// TIA Portal V16 export
// export: Created 2021-11-12T13:31:09.8537827Z, ExportSetting WithDefaults, DisplayName Totally Integrated Automation Portal, DisplayVersion V16 Update 3, DisplayName TIA Portal Version Control Interface, DisplayVersion V16 Update 2, DisplayName TIA Portal Openness, DisplayVersion V16 Update 3, DisplayName SINAMICS Startdrive Advanced, DisplayVersion V16 Update 5, DisplayName SINAMICS Startdrive G130, G150, S120, S150, SINAMICS MV, S210, DisplayVersion V16 Update 5, DisplayName SINAMICS Startdrive G110M, G120, G120C, G120D, G120P, G115D, DisplayVersion V16 Update 5, DisplayName STEP 7 Professional, DisplayVersion V16 Update 3, DisplayName STEP 7 Safety, DisplayVersion V16, DisplayName WinCC UA Professional, DisplayVersion V16 Update 3
FUNCTION_BLOCK "Sfty_Outputs"   // FB74, F_LAD
{ S7_Optimized_Access := 'TRUE' }
VERSION : 0.1
// stored: AutoNumber true, IsIECCheckEnabled false, UDAEnableTagReadback false
   VAR
      "SF_100UH01-KF51_A1" : FDBACK;
      "SF_400UH01-KF51_A1" : FDBACK;
      "SF_100UH01-KF52_A1" : FDBACK;
      "SF_100UH01-KF53_A1" : FDBACK;
   END_VAR
   VAR_TEMP
      TB1EstopZ100 : Bool;   // Estop ok zone 100
      TB1EstopZ200 : Bool;   // Estop ok zone 200
      TB1EstopZ300 : Bool;   // Estop ok zone 300
      TB1EstopZ400 : Bool;   // Estop ok zone 400
      TB1FenceZ101 : Bool;   // Doors locked zone 101
      TB1FenceZ102 : Bool;   // Doors locked zone 102
      TB1FenceZ103 : Bool;   // Doors locked zone 103
      TB1FenceZ104 : Bool;   // Doors locked zone 104
      TB1FenceZ105 : Bool;   // Doors locked zone 105
      TB1FenceZ200 : Bool;   // Doors locked zone 200
      TB1FenceZ300 : Bool;   // Doors locked zone 300
      TB1FenceZ400 : Bool;   // Doors locked zone 400
      TB1Bin : Bool;   // Commissioning
   END_VAR
BEGIN

REGION Network 1: *************** Estop ***************
END_REGION

REGION Network 2: All estops in zone 100 ok
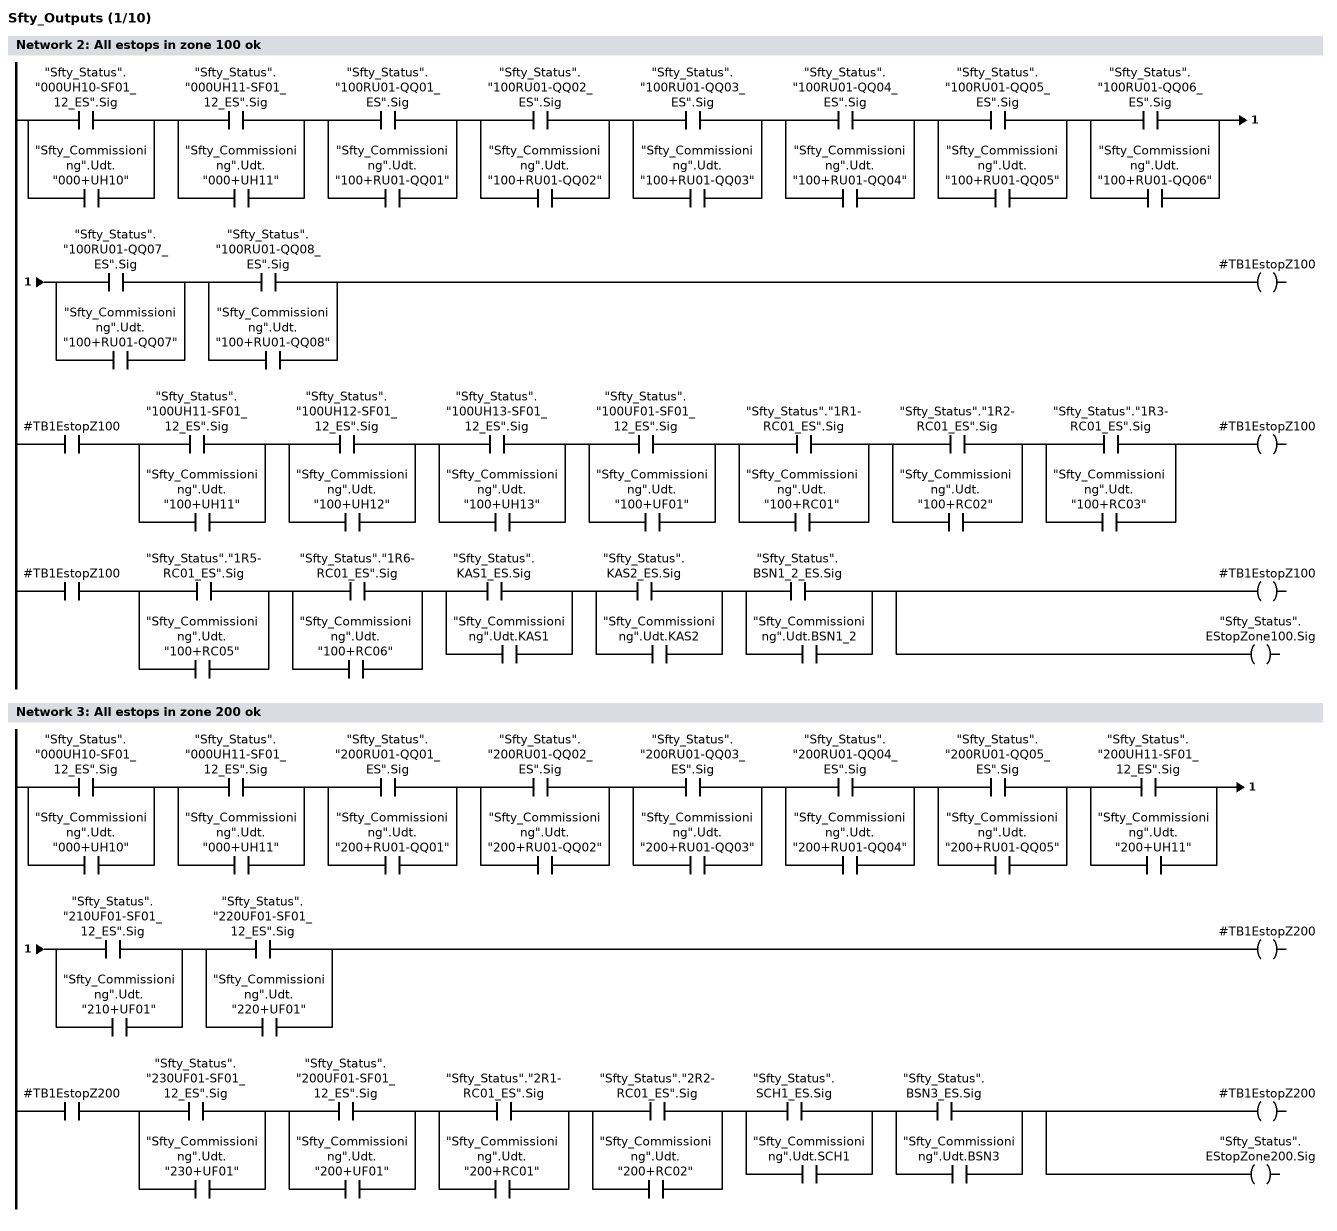
   RUNG wire#powerrail
      Contact( "Sfty_Status"."000UH10-SF01_12_ES".Sig )
      wire#w1
      Contact( "Sfty_Status"."000UH11-SF01_12_ES".Sig )
      wire#w2
      Contact( "Sfty_Status"."100RU01-QQ01_ES".Sig )
      wire#w3
      Contact( "Sfty_Status"."100RU01-QQ02_ES".Sig )
      wire#w4
      Contact( "Sfty_Status"."100RU01-QQ03_ES".Sig )
      wire#w5
      Contact( "Sfty_Status"."100RU01-QQ04_ES".Sig )
      wire#w6
      Contact( "Sfty_Status"."100RU01-QQ05_ES".Sig )
      wire#w7
      Contact( "Sfty_Status"."100RU01-QQ06_ES".Sig )
      wire#w8
      Contact( "Sfty_Status"."100RU01-QQ07_ES".Sig )
      wire#w9
      Contact( "Sfty_Status"."100RU01-QQ08_ES".Sig )
      wire#w10
      Coil( #TB1EstopZ100 )
   END_RUNG
   RUNG wire#powerrail
      Contact( "Sfty_Commissioning".Udt."000+UH10" )
   END_RUNG wire#w1
   RUNG wire#w1
      Contact( "Sfty_Commissioning".Udt."000+UH11" )
   END_RUNG wire#w2
   RUNG wire#w2
      Contact( "Sfty_Commissioning".Udt."100+RU01-QQ01" )
   END_RUNG wire#w3
   RUNG wire#w3
      Contact( "Sfty_Commissioning".Udt."100+RU01-QQ02" )
   END_RUNG wire#w4
   RUNG wire#w4
      Contact( "Sfty_Commissioning".Udt."100+RU01-QQ03" )
   END_RUNG wire#w5
   RUNG wire#w5
      Contact( "Sfty_Commissioning".Udt."100+RU01-QQ04" )
   END_RUNG wire#w6
   RUNG wire#w6
      Contact( "Sfty_Commissioning".Udt."100+RU01-QQ05" )
   END_RUNG wire#w7
   RUNG wire#w7
      Contact( "Sfty_Commissioning".Udt."100+RU01-QQ06" )
   END_RUNG wire#w8
   RUNG wire#w8
      Contact( "Sfty_Commissioning".Udt."100+RU01-QQ07" )
   END_RUNG wire#w9
   RUNG wire#w9
      Contact( "Sfty_Commissioning".Udt."100+RU01-QQ08" )
   END_RUNG wire#w10
   RUNG wire#powerrail
      Contact( #TB1EstopZ100 )
      wire#w11
      Contact( "Sfty_Status"."100UH11-SF01_12_ES".Sig )
      wire#w12
      Contact( "Sfty_Status"."100UH12-SF01_12_ES".Sig )
      wire#w13
      Contact( "Sfty_Status"."100UH13-SF01_12_ES".Sig )
      wire#w14
      Contact( "Sfty_Status"."100UF01-SF01_12_ES".Sig )
      wire#w15
      Contact( "Sfty_Status"."1R1-RC01_ES".Sig )
      wire#w16
      Contact( "Sfty_Status"."1R2-RC01_ES".Sig )
      wire#w17
      Contact( "Sfty_Status"."1R3-RC01_ES".Sig )
      wire#w18
      Coil( #TB1EstopZ100 )
   END_RUNG
   RUNG wire#w11
      Contact( "Sfty_Commissioning".Udt."100+UH11" )
   END_RUNG wire#w12
   RUNG wire#w12
      Contact( "Sfty_Commissioning".Udt."100+UH12" )
   END_RUNG wire#w13
   RUNG wire#w13
      Contact( "Sfty_Commissioning".Udt."100+UH13" )
   END_RUNG wire#w14
   RUNG wire#w14
      Contact( "Sfty_Commissioning".Udt."100+UF01" )
   END_RUNG wire#w15
   RUNG wire#w15
      Contact( "Sfty_Commissioning".Udt."100+RC01" )
   END_RUNG wire#w16
   RUNG wire#w16
      Contact( "Sfty_Commissioning".Udt."100+RC02" )
   END_RUNG wire#w17
   RUNG wire#w17
      Contact( "Sfty_Commissioning".Udt."100+RC03" )
   END_RUNG wire#w18
   RUNG wire#powerrail
      Contact( #TB1EstopZ100 )
      wire#w19
      Contact( "Sfty_Status"."1R5-RC01_ES".Sig )
      wire#w20
      Contact( "Sfty_Status"."1R6-RC01_ES".Sig )
      wire#w21
      Contact( "Sfty_Status".KAS1_ES.Sig )
      wire#w22
      Contact( "Sfty_Status".KAS2_ES.Sig )
      wire#w23
      Contact( "Sfty_Status".BSN1_2_ES.Sig )
      wire#w24
      Coil( #TB1EstopZ100 )
   END_RUNG
   RUNG wire#w19
      Contact( "Sfty_Commissioning".Udt."100+RC05" )
   END_RUNG wire#w20
   RUNG wire#w20
      Contact( "Sfty_Commissioning".Udt."100+RC06" )
   END_RUNG wire#w21
   RUNG wire#w21
      Contact( "Sfty_Commissioning".Udt.KAS1 )
   END_RUNG wire#w22
   RUNG wire#w22
      Contact( "Sfty_Commissioning".Udt.KAS2 )
   END_RUNG wire#w23
   RUNG wire#w23
      Contact( "Sfty_Commissioning".Udt.BSN1_2 )
   END_RUNG wire#w24
   RUNG wire#w24
      Coil( "Sfty_Status".EStopZone100.Sig )
   END_RUNG
   // the same network as SCL:
   #TB1EstopZ100 := ("Sfty_Status"."000UH10-SF01_12_ES".Sig OR "Sfty_Commissioning".Udt."000+UH10") AND ("Sfty_Status"."000UH11-SF01_12_ES".Sig OR "Sfty_Commissioning".Udt."000+UH11") AND ("Sfty_Status"."100RU01-QQ01_ES".Sig OR "Sfty_Commissioning".Udt."100+RU01-QQ01") AND ("Sfty_Status"."100RU01-QQ02_ES".Sig OR "Sfty_Commissioning".Udt."100+RU01-QQ02") AND ("Sfty_Status"."100RU01-QQ03_ES".Sig OR "Sfty_Commissioning".Udt."100+RU01-QQ03") AND ("Sfty_Status"."100RU01-QQ04_ES".Sig OR "Sfty_Commissioning".Udt."100+RU01-QQ04") AND ("Sfty_Status"."100RU01-QQ05_ES".Sig OR "Sfty_Commissioning".Udt."100+RU01-QQ05") AND ("Sfty_Status"."100RU01-QQ06_ES".Sig OR "Sfty_Commissioning".Udt."100+RU01-QQ06") AND ("Sfty_Status"."100RU01-QQ07_ES".Sig OR "Sfty_Commissioning".Udt."100+RU01-QQ07") AND ("Sfty_Status"."100RU01-QQ08_ES".Sig OR "Sfty_Commissioning".Udt."100+RU01-QQ08");
   #TB1EstopZ100 := #TB1EstopZ100 AND ("Sfty_Status"."100UH11-SF01_12_ES".Sig OR "Sfty_Commissioning".Udt."100+UH11") AND ("Sfty_Status"."100UH12-SF01_12_ES".Sig OR "Sfty_Commissioning".Udt."100+UH12") AND ("Sfty_Status"."100UH13-SF01_12_ES".Sig OR "Sfty_Commissioning".Udt."100+UH13") AND ("Sfty_Status"."100UF01-SF01_12_ES".Sig OR "Sfty_Commissioning".Udt."100+UF01") AND ("Sfty_Status"."1R1-RC01_ES".Sig OR "Sfty_Commissioning".Udt."100+RC01") AND ("Sfty_Status"."1R2-RC01_ES".Sig OR "Sfty_Commissioning".Udt."100+RC02") AND ("Sfty_Status"."1R3-RC01_ES".Sig OR "Sfty_Commissioning".Udt."100+RC03");
   #TB1EstopZ100 := #TB1EstopZ100 AND ("Sfty_Status"."1R5-RC01_ES".Sig OR "Sfty_Commissioning".Udt."100+RC05") AND ("Sfty_Status"."1R6-RC01_ES".Sig OR "Sfty_Commissioning".Udt."100+RC06") AND ("Sfty_Status".KAS1_ES.Sig OR "Sfty_Commissioning".Udt.KAS1) AND ("Sfty_Status".KAS2_ES.Sig OR "Sfty_Commissioning".Udt.KAS2) AND ("Sfty_Status".BSN1_2_ES.Sig OR "Sfty_Commissioning".Udt.BSN1_2);
   "Sfty_Status".EStopZone100.Sig := #TB1EstopZ100;
END_REGION

REGION Network 3: All estops in zone 200 ok
   RUNG wire#powerrail
      Contact( "Sfty_Status"."000UH10-SF01_12_ES".Sig )
      wire#w1
      Contact( "Sfty_Status"."000UH11-SF01_12_ES".Sig )
      wire#w2
      Contact( "Sfty_Status"."200RU01-QQ01_ES".Sig )
      wire#w3
      Contact( "Sfty_Status"."200RU01-QQ02_ES".Sig )
      wire#w4
      Contact( "Sfty_Status"."200RU01-QQ03_ES".Sig )
      wire#w5
      Contact( "Sfty_Status"."200RU01-QQ04_ES".Sig )
      wire#w6
      Contact( "Sfty_Status"."200RU01-QQ05_ES".Sig )
      wire#w7
      Contact( "Sfty_Status"."200UH11-SF01_12_ES".Sig )
      wire#w8
      Contact( "Sfty_Status"."210UF01-SF01_12_ES".Sig )
      wire#w9
      Contact( "Sfty_Status"."220UF01-SF01_12_ES".Sig )
      wire#w10
      Coil( #TB1EstopZ200 )
   END_RUNG
   RUNG wire#powerrail
      Contact( "Sfty_Commissioning".Udt."000+UH10" )
   END_RUNG wire#w1
   RUNG wire#w1
      Contact( "Sfty_Commissioning".Udt."000+UH11" )
   END_RUNG wire#w2
   RUNG wire#w2
      Contact( "Sfty_Commissioning".Udt."200+RU01-QQ01" )
   END_RUNG wire#w3
   RUNG wire#w3
      Contact( "Sfty_Commissioning".Udt."200+RU01-QQ02" )
   END_RUNG wire#w4
   RUNG wire#w4
      Contact( "Sfty_Commissioning".Udt."200+RU01-QQ03" )
   END_RUNG wire#w5
   RUNG wire#w5
      Contact( "Sfty_Commissioning".Udt."200+RU01-QQ04" )
   END_RUNG wire#w6
   RUNG wire#w6
      Contact( "Sfty_Commissioning".Udt."200+RU01-QQ05" )
   END_RUNG wire#w7
   RUNG wire#w7
      Contact( "Sfty_Commissioning".Udt."200+UH11" )
   END_RUNG wire#w8
   RUNG wire#w8
      Contact( "Sfty_Commissioning".Udt."210+UF01" )
   END_RUNG wire#w9
   RUNG wire#w9
      Contact( "Sfty_Commissioning".Udt."220+UF01" )
   END_RUNG wire#w10
   RUNG wire#powerrail
      Contact( #TB1EstopZ200 )
      wire#w11
      Contact( "Sfty_Status"."230UF01-SF01_12_ES".Sig )
      wire#w12
      Contact( "Sfty_Status"."200UF01-SF01_12_ES".Sig )
      wire#w13
      Contact( "Sfty_Status"."2R1-RC01_ES".Sig )
      wire#w14
      Contact( "Sfty_Status"."2R2-RC01_ES".Sig )
      wire#w15
      Contact( "Sfty_Status".SCH1_ES.Sig )
      wire#w16
      Contact( "Sfty_Status".BSN3_ES.Sig )
      wire#w17
      Coil( #TB1EstopZ200 )
   END_RUNG
   RUNG wire#w11
      Contact( "Sfty_Commissioning".Udt."230+UF01" )
   END_RUNG wire#w12
   RUNG wire#w12
      Contact( "Sfty_Commissioning".Udt."200+UF01" )
   END_RUNG wire#w13
   RUNG wire#w13
      Contact( "Sfty_Commissioning".Udt."200+RC01" )
   END_RUNG wire#w14
   RUNG wire#w14
      Contact( "Sfty_Commissioning".Udt."200+RC02" )
   END_RUNG wire#w15
   RUNG wire#w15
      Contact( "Sfty_Commissioning".Udt.SCH1 )
   END_RUNG wire#w16
   RUNG wire#w16
      Contact( "Sfty_Commissioning".Udt.BSN3 )
   END_RUNG wire#w17
   RUNG wire#w17
      Coil( "Sfty_Status".EStopZone200.Sig )
   END_RUNG
   // the same network as SCL:
   #TB1EstopZ200 := ("Sfty_Status"."000UH10-SF01_12_ES".Sig OR "Sfty_Commissioning".Udt."000+UH10") AND ("Sfty_Status"."000UH11-SF01_12_ES".Sig OR "Sfty_Commissioning".Udt."000+UH11") AND ("Sfty_Status"."200RU01-QQ01_ES".Sig OR "Sfty_Commissioning".Udt."200+RU01-QQ01") AND ("Sfty_Status"."200RU01-QQ02_ES".Sig OR "Sfty_Commissioning".Udt."200+RU01-QQ02") AND ("Sfty_Status"."200RU01-QQ03_ES".Sig OR "Sfty_Commissioning".Udt."200+RU01-QQ03") AND ("Sfty_Status"."200RU01-QQ04_ES".Sig OR "Sfty_Commissioning".Udt."200+RU01-QQ04") AND ("Sfty_Status"."200RU01-QQ05_ES".Sig OR "Sfty_Commissioning".Udt."200+RU01-QQ05") AND ("Sfty_Status"."200UH11-SF01_12_ES".Sig OR "Sfty_Commissioning".Udt."200+UH11") AND ("Sfty_Status"."210UF01-SF01_12_ES".Sig OR "Sfty_Commissioning".Udt."210+UF01") AND ("Sfty_Status"."220UF01-SF01_12_ES".Sig OR "Sfty_Commissioning".Udt."220+UF01");
   #TB1EstopZ200 := #TB1EstopZ200 AND ("Sfty_Status"."230UF01-SF01_12_ES".Sig OR "Sfty_Commissioning".Udt."230+UF01") AND ("Sfty_Status"."200UF01-SF01_12_ES".Sig OR "Sfty_Commissioning".Udt."200+UF01") AND ("Sfty_Status"."2R1-RC01_ES".Sig OR "Sfty_Commissioning".Udt."200+RC01") AND ("Sfty_Status"."2R2-RC01_ES".Sig OR "Sfty_Commissioning".Udt."200+RC02") AND ("Sfty_Status".SCH1_ES.Sig OR "Sfty_Commissioning".Udt.SCH1) AND ("Sfty_Status".BSN3_ES.Sig OR "Sfty_Commissioning".Udt.BSN3);
   "Sfty_Status".EStopZone200.Sig := #TB1EstopZ200;
END_REGION

REGION Network 4: All estops in zone 300 ok
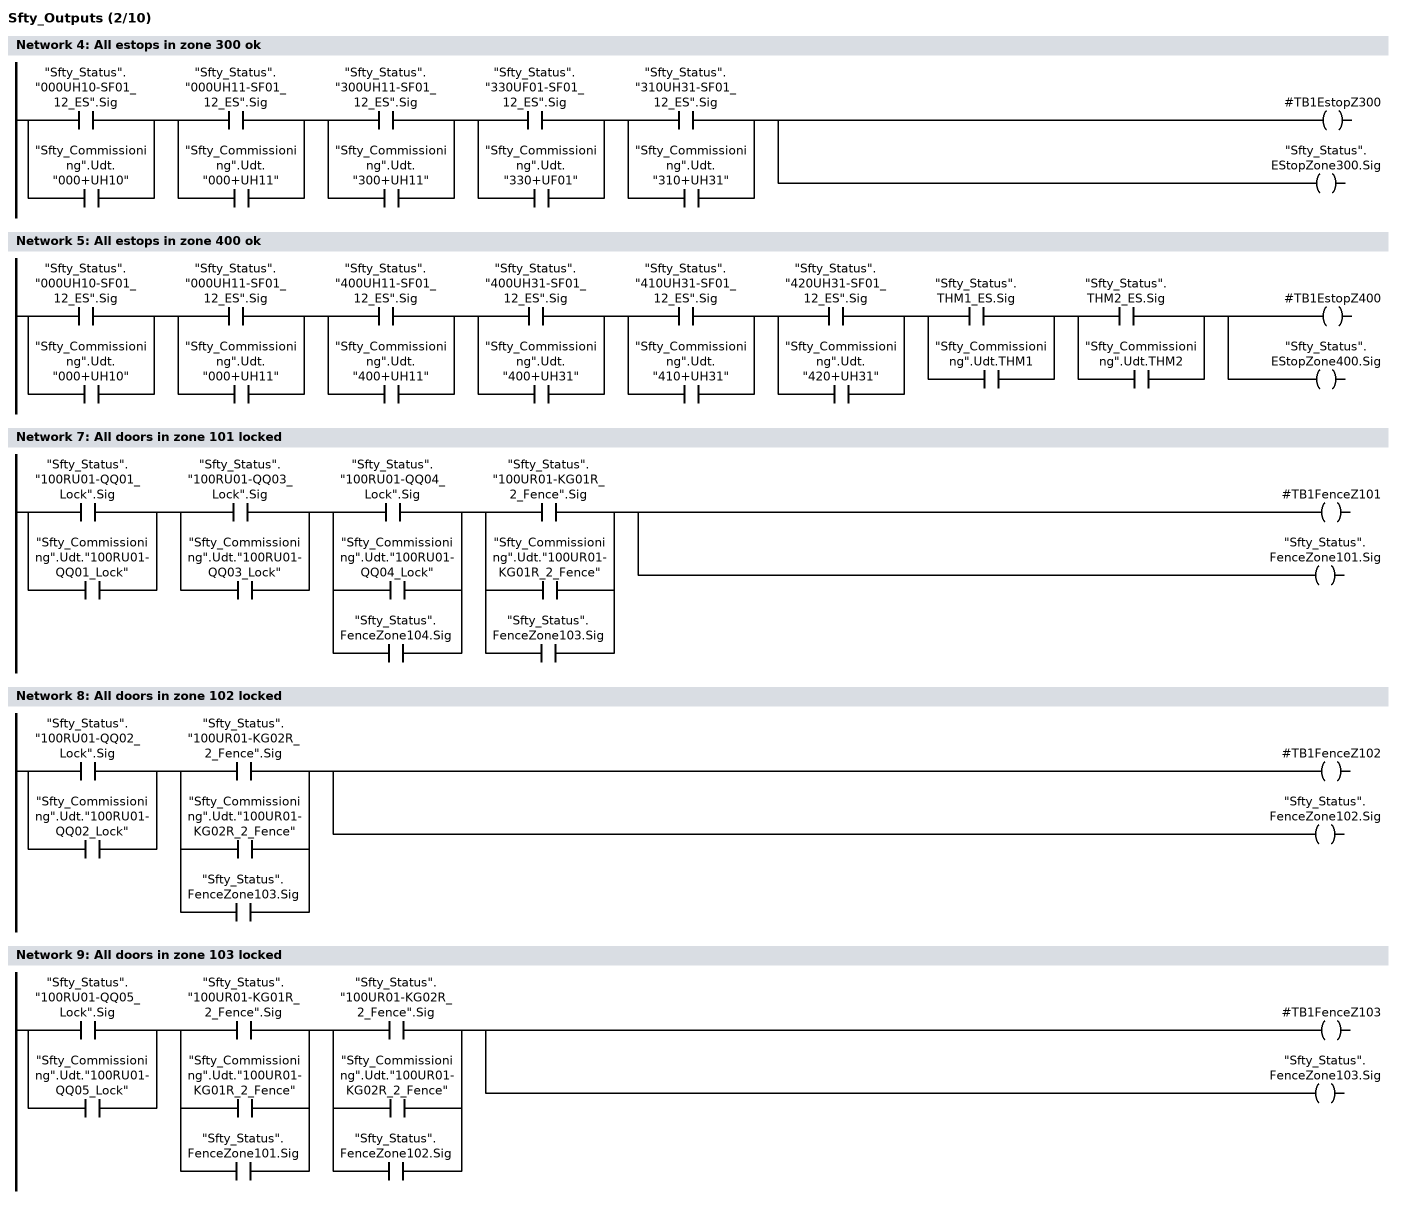
   RUNG wire#powerrail
      Contact( "Sfty_Status"."000UH10-SF01_12_ES".Sig )
      wire#w1
      Contact( "Sfty_Status"."000UH11-SF01_12_ES".Sig )
      wire#w2
      Contact( "Sfty_Status"."300UH11-SF01_12_ES".Sig )
      wire#w3
      Contact( "Sfty_Status"."330UF01-SF01_12_ES".Sig )
      wire#w4
      Contact( "Sfty_Status"."310UH31-SF01_12_ES".Sig )
      wire#w5
      Coil( #TB1EstopZ300 )
   END_RUNG
   RUNG wire#powerrail
      Contact( "Sfty_Commissioning".Udt."000+UH10" )
   END_RUNG wire#w1
   RUNG wire#w1
      Contact( "Sfty_Commissioning".Udt."000+UH11" )
   END_RUNG wire#w2
   RUNG wire#w2
      Contact( "Sfty_Commissioning".Udt."300+UH11" )
   END_RUNG wire#w3
   RUNG wire#w3
      Contact( "Sfty_Commissioning".Udt."330+UF01" )
   END_RUNG wire#w4
   RUNG wire#w4
      Contact( "Sfty_Commissioning".Udt."310+UH31" )
   END_RUNG wire#w5
   RUNG wire#w5
      Coil( "Sfty_Status".EStopZone300.Sig )
   END_RUNG
   // the same network as SCL:
   #TB1EstopZ300 := ("Sfty_Status"."000UH10-SF01_12_ES".Sig OR "Sfty_Commissioning".Udt."000+UH10") AND ("Sfty_Status"."000UH11-SF01_12_ES".Sig OR "Sfty_Commissioning".Udt."000+UH11") AND ("Sfty_Status"."300UH11-SF01_12_ES".Sig OR "Sfty_Commissioning".Udt."300+UH11") AND ("Sfty_Status"."330UF01-SF01_12_ES".Sig OR "Sfty_Commissioning".Udt."330+UF01") AND ("Sfty_Status"."310UH31-SF01_12_ES".Sig OR "Sfty_Commissioning".Udt."310+UH31");
   "Sfty_Status".EStopZone300.Sig := #TB1EstopZ300;
END_REGION

REGION Network 5: All estops in zone 400 ok
   RUNG wire#powerrail
      Contact( "Sfty_Status"."000UH10-SF01_12_ES".Sig )
      wire#w1
      Contact( "Sfty_Status"."000UH11-SF01_12_ES".Sig )
      wire#w2
      Contact( "Sfty_Status"."400UH11-SF01_12_ES".Sig )
      wire#w3
      Contact( "Sfty_Status"."400UH31-SF01_12_ES".Sig )
      wire#w4
      Contact( "Sfty_Status"."410UH31-SF01_12_ES".Sig )
      wire#w5
      Contact( "Sfty_Status"."420UH31-SF01_12_ES".Sig )
      wire#w6
      Contact( "Sfty_Status".THM1_ES.Sig )
      wire#w7
      Contact( "Sfty_Status".THM2_ES.Sig )
      wire#w8
      Coil( #TB1EstopZ400 )
   END_RUNG
   RUNG wire#powerrail
      Contact( "Sfty_Commissioning".Udt."000+UH10" )
   END_RUNG wire#w1
   RUNG wire#w1
      Contact( "Sfty_Commissioning".Udt."000+UH11" )
   END_RUNG wire#w2
   RUNG wire#w2
      Contact( "Sfty_Commissioning".Udt."400+UH11" )
   END_RUNG wire#w3
   RUNG wire#w3
      Contact( "Sfty_Commissioning".Udt."400+UH31" )
   END_RUNG wire#w4
   RUNG wire#w4
      Contact( "Sfty_Commissioning".Udt."410+UH31" )
   END_RUNG wire#w5
   RUNG wire#w5
      Contact( "Sfty_Commissioning".Udt."420+UH31" )
   END_RUNG wire#w6
   RUNG wire#w6
      Contact( "Sfty_Commissioning".Udt.THM1 )
   END_RUNG wire#w7
   RUNG wire#w7
      Contact( "Sfty_Commissioning".Udt.THM2 )
   END_RUNG wire#w8
   RUNG wire#w8
      Coil( "Sfty_Status".EStopZone400.Sig )
   END_RUNG
   // the same network as SCL:
   #TB1EstopZ400 := ("Sfty_Status"."000UH10-SF01_12_ES".Sig OR "Sfty_Commissioning".Udt."000+UH10") AND ("Sfty_Status"."000UH11-SF01_12_ES".Sig OR "Sfty_Commissioning".Udt."000+UH11") AND ("Sfty_Status"."400UH11-SF01_12_ES".Sig OR "Sfty_Commissioning".Udt."400+UH11") AND ("Sfty_Status"."400UH31-SF01_12_ES".Sig OR "Sfty_Commissioning".Udt."400+UH31") AND ("Sfty_Status"."410UH31-SF01_12_ES".Sig OR "Sfty_Commissioning".Udt."410+UH31") AND ("Sfty_Status"."420UH31-SF01_12_ES".Sig OR "Sfty_Commissioning".Udt."420+UH31") AND ("Sfty_Status".THM1_ES.Sig OR "Sfty_Commissioning".Udt.THM1) AND ("Sfty_Status".THM2_ES.Sig OR "Sfty_Commissioning".Udt.THM2);
   "Sfty_Status".EStopZone400.Sig := #TB1EstopZ400;
END_REGION

REGION Network 6: *************** Fence ***************
END_REGION

REGION Network 7: All doors in zone 101 locked
   RUNG wire#powerrail
      Contact( "Sfty_Status"."100RU01-QQ01_Lock".Sig )
      wire#w1
      Contact( "Sfty_Status"."100RU01-QQ03_Lock".Sig )
      wire#w2
      Contact( "Sfty_Status"."100RU01-QQ04_Lock".Sig )
      wire#w3
      Contact( "Sfty_Status"."100UR01-KG01R_2_Fence".Sig )
      wire#w4
      Coil( #TB1FenceZ101 )
   END_RUNG
   RUNG wire#powerrail
      Contact( "Sfty_Commissioning".Udt."100RU01-QQ01_Lock" )
   END_RUNG wire#w1
   RUNG wire#w1
      Contact( "Sfty_Commissioning".Udt."100RU01-QQ03_Lock" )
   END_RUNG wire#w2
   RUNG wire#w2
      Contact( "Sfty_Commissioning".Udt."100RU01-QQ04_Lock" )
   END_RUNG wire#w3
   RUNG wire#w2
      Contact( "Sfty_Status".FenceZone104.Sig )
   END_RUNG wire#w3
   RUNG wire#w3
      Contact( "Sfty_Commissioning".Udt."100UR01-KG01R_2_Fence" )
   END_RUNG wire#w4
   RUNG wire#w3
      Contact( "Sfty_Status".FenceZone103.Sig )
   END_RUNG wire#w4
   RUNG wire#w4
      Coil( "Sfty_Status".FenceZone101.Sig )
   END_RUNG
   // the same network as SCL:
   #TB1FenceZ101 := ("Sfty_Status"."100RU01-QQ01_Lock".Sig OR "Sfty_Commissioning".Udt."100RU01-QQ01_Lock") AND ("Sfty_Status"."100RU01-QQ03_Lock".Sig OR "Sfty_Commissioning".Udt."100RU01-QQ03_Lock") AND ("Sfty_Status"."100RU01-QQ04_Lock".Sig OR "Sfty_Commissioning".Udt."100RU01-QQ04_Lock" OR "Sfty_Status".FenceZone104.Sig) AND ("Sfty_Status"."100UR01-KG01R_2_Fence".Sig OR "Sfty_Commissioning".Udt."100UR01-KG01R_2_Fence" OR "Sfty_Status".FenceZone103.Sig);
   "Sfty_Status".FenceZone101.Sig := #TB1FenceZ101;
END_REGION

REGION Network 8: All doors in zone 102 locked
   RUNG wire#powerrail
      Contact( "Sfty_Status"."100RU01-QQ02_Lock".Sig )
      wire#w1
      Contact( "Sfty_Status"."100UR01-KG02R_2_Fence".Sig )
      wire#w2
      Coil( #TB1FenceZ102 )
   END_RUNG
   RUNG wire#powerrail
      Contact( "Sfty_Commissioning".Udt."100RU01-QQ02_Lock" )
   END_RUNG wire#w1
   RUNG wire#w1
      Contact( "Sfty_Commissioning".Udt."100UR01-KG02R_2_Fence" )
   END_RUNG wire#w2
   RUNG wire#w1
      Contact( "Sfty_Status".FenceZone103.Sig )
   END_RUNG wire#w2
   RUNG wire#w2
      Coil( "Sfty_Status".FenceZone102.Sig )
   END_RUNG
   // the same network as SCL:
   #TB1FenceZ102 := ("Sfty_Status"."100RU01-QQ02_Lock".Sig OR "Sfty_Commissioning".Udt."100RU01-QQ02_Lock") AND ("Sfty_Status"."100UR01-KG02R_2_Fence".Sig OR "Sfty_Commissioning".Udt."100UR01-KG02R_2_Fence" OR "Sfty_Status".FenceZone103.Sig);
   "Sfty_Status".FenceZone102.Sig := #TB1FenceZ102;
END_REGION

REGION Network 9: All doors in zone 103 locked
   RUNG wire#powerrail
      Contact( "Sfty_Status"."100RU01-QQ05_Lock".Sig )
      wire#w1
      Contact( "Sfty_Status"."100UR01-KG01R_2_Fence".Sig )
      wire#w2
      Contact( "Sfty_Status"."100UR01-KG02R_2_Fence".Sig )
      wire#w3
      Coil( #TB1FenceZ103 )
   END_RUNG
   RUNG wire#powerrail
      Contact( "Sfty_Commissioning".Udt."100RU01-QQ05_Lock" )
   END_RUNG wire#w1
   RUNG wire#w1
      Contact( "Sfty_Commissioning".Udt."100UR01-KG01R_2_Fence" )
   END_RUNG wire#w2
   RUNG wire#w1
      Contact( "Sfty_Status".FenceZone101.Sig )
   END_RUNG wire#w2
   RUNG wire#w2
      Contact( "Sfty_Commissioning".Udt."100UR01-KG02R_2_Fence" )
   END_RUNG wire#w3
   RUNG wire#w2
      Contact( "Sfty_Status".FenceZone102.Sig )
   END_RUNG wire#w3
   RUNG wire#w3
      Coil( "Sfty_Status".FenceZone103.Sig )
   END_RUNG
   // the same network as SCL:
   #TB1FenceZ103 := ("Sfty_Status"."100RU01-QQ05_Lock".Sig OR "Sfty_Commissioning".Udt."100RU01-QQ05_Lock") AND ("Sfty_Status"."100UR01-KG01R_2_Fence".Sig OR "Sfty_Commissioning".Udt."100UR01-KG01R_2_Fence" OR "Sfty_Status".FenceZone101.Sig) AND ("Sfty_Status"."100UR01-KG02R_2_Fence".Sig OR "Sfty_Commissioning".Udt."100UR01-KG02R_2_Fence" OR "Sfty_Status".FenceZone102.Sig);
   "Sfty_Status".FenceZone103.Sig := #TB1FenceZ103;
END_REGION

REGION Network 10: All doors in zone 104 locked
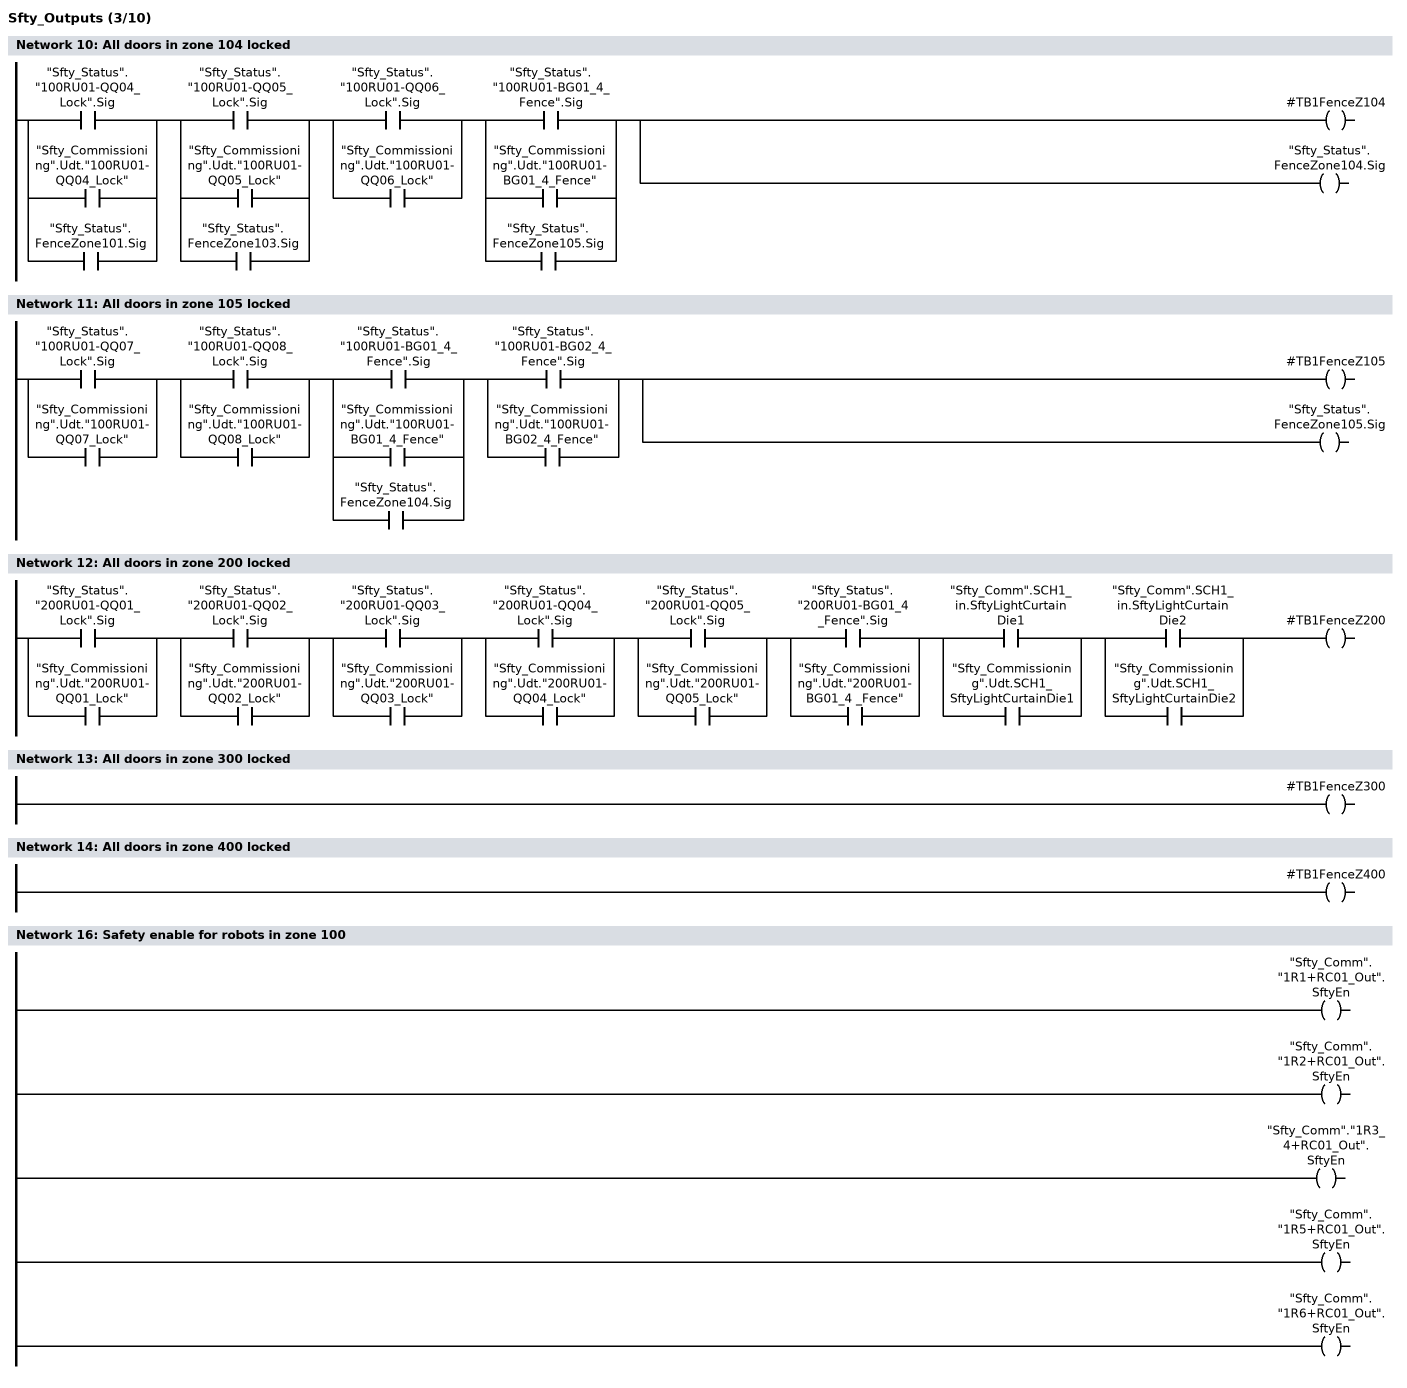
   RUNG wire#powerrail
      Contact( "Sfty_Status"."100RU01-QQ04_Lock".Sig )
      wire#w1
      Contact( "Sfty_Status"."100RU01-QQ05_Lock".Sig )
      wire#w2
      Contact( "Sfty_Status"."100RU01-QQ06_Lock".Sig )
      wire#w3
      Contact( "Sfty_Status"."100RU01-BG01_4_Fence".Sig )
      wire#w4
      Coil( #TB1FenceZ104 )
   END_RUNG
   RUNG wire#powerrail
      Contact( "Sfty_Commissioning".Udt."100RU01-QQ04_Lock" )
   END_RUNG wire#w1
   RUNG wire#powerrail
      Contact( "Sfty_Status".FenceZone101.Sig )
   END_RUNG wire#w1
   RUNG wire#w1
      Contact( "Sfty_Commissioning".Udt."100RU01-QQ05_Lock" )
   END_RUNG wire#w2
   RUNG wire#w1
      Contact( "Sfty_Status".FenceZone103.Sig )
   END_RUNG wire#w2
   RUNG wire#w2
      Contact( "Sfty_Commissioning".Udt."100RU01-QQ06_Lock" )
   END_RUNG wire#w3
   RUNG wire#w3
      Contact( "Sfty_Commissioning".Udt."100RU01-BG01_4_Fence" )
   END_RUNG wire#w4
   RUNG wire#w3
      Contact( "Sfty_Status".FenceZone105.Sig )
   END_RUNG wire#w4
   RUNG wire#w4
      Coil( "Sfty_Status".FenceZone104.Sig )
   END_RUNG
   // the same network as SCL:
   #TB1FenceZ104 := ("Sfty_Status"."100RU01-QQ04_Lock".Sig OR "Sfty_Commissioning".Udt."100RU01-QQ04_Lock" OR "Sfty_Status".FenceZone101.Sig) AND ("Sfty_Status"."100RU01-QQ05_Lock".Sig OR "Sfty_Commissioning".Udt."100RU01-QQ05_Lock" OR "Sfty_Status".FenceZone103.Sig) AND ("Sfty_Status"."100RU01-QQ06_Lock".Sig OR "Sfty_Commissioning".Udt."100RU01-QQ06_Lock") AND ("Sfty_Status"."100RU01-BG01_4_Fence".Sig OR "Sfty_Commissioning".Udt."100RU01-BG01_4_Fence" OR "Sfty_Status".FenceZone105.Sig);
   "Sfty_Status".FenceZone104.Sig := #TB1FenceZ104;
END_REGION

REGION Network 11: All doors in zone 105 locked
   RUNG wire#powerrail
      Contact( "Sfty_Status"."100RU01-QQ07_Lock".Sig )
      wire#w1
      Contact( "Sfty_Status"."100RU01-QQ08_Lock".Sig )
      wire#w2
      Contact( "Sfty_Status"."100RU01-BG01_4_Fence".Sig )
      wire#w3
      Contact( "Sfty_Status"."100RU01-BG02_4_Fence".Sig )
      wire#w4
      Coil( #TB1FenceZ105 )
   END_RUNG
   RUNG wire#powerrail
      Contact( "Sfty_Commissioning".Udt."100RU01-QQ07_Lock" )
   END_RUNG wire#w1
   RUNG wire#w1
      Contact( "Sfty_Commissioning".Udt."100RU01-QQ08_Lock" )
   END_RUNG wire#w2
   RUNG wire#w2
      Contact( "Sfty_Commissioning".Udt."100RU01-BG01_4_Fence" )
   END_RUNG wire#w3
   RUNG wire#w2
      Contact( "Sfty_Status".FenceZone104.Sig )
   END_RUNG wire#w3
   RUNG wire#w3
      Contact( "Sfty_Commissioning".Udt."100RU01-BG02_4_Fence" )
   END_RUNG wire#w4
   RUNG wire#w4
      Coil( "Sfty_Status".FenceZone105.Sig )
   END_RUNG
   // the same network as SCL:
   #TB1FenceZ105 := ("Sfty_Status"."100RU01-QQ07_Lock".Sig OR "Sfty_Commissioning".Udt."100RU01-QQ07_Lock") AND ("Sfty_Status"."100RU01-QQ08_Lock".Sig OR "Sfty_Commissioning".Udt."100RU01-QQ08_Lock") AND ("Sfty_Status"."100RU01-BG01_4_Fence".Sig OR "Sfty_Commissioning".Udt."100RU01-BG01_4_Fence" OR "Sfty_Status".FenceZone104.Sig) AND ("Sfty_Status"."100RU01-BG02_4_Fence".Sig OR "Sfty_Commissioning".Udt."100RU01-BG02_4_Fence");
   "Sfty_Status".FenceZone105.Sig := #TB1FenceZ105;
END_REGION

REGION Network 12: All doors in zone 200 locked
   RUNG wire#powerrail
      Contact( "Sfty_Status"."200RU01-QQ01_Lock".Sig )
      wire#w1
      Contact( "Sfty_Status"."200RU01-QQ02_Lock".Sig )
      wire#w2
      Contact( "Sfty_Status"."200RU01-QQ03_Lock".Sig )
      wire#w3
      Contact( "Sfty_Status"."200RU01-QQ04_Lock".Sig )
      wire#w4
      Contact( "Sfty_Status"."200RU01-QQ05_Lock".Sig )
      wire#w5
      Contact( "Sfty_Status"."200RU01-BG01_4 _Fence".Sig )
      wire#w6
      Contact( "Sfty_Comm".SCH1_in.SftyLightCurtainDie1 )
      wire#w7
      Contact( "Sfty_Comm".SCH1_in.SftyLightCurtainDie2 )
      wire#w8
      Coil( #TB1FenceZ200 )
   END_RUNG
   RUNG wire#powerrail
      Contact( "Sfty_Commissioning".Udt."200RU01-QQ01_Lock" )
   END_RUNG wire#w1
   RUNG wire#w1
      Contact( "Sfty_Commissioning".Udt."200RU01-QQ02_Lock" )
   END_RUNG wire#w2
   RUNG wire#w2
      Contact( "Sfty_Commissioning".Udt."200RU01-QQ03_Lock" )
   END_RUNG wire#w3
   RUNG wire#w3
      Contact( "Sfty_Commissioning".Udt."200RU01-QQ04_Lock" )
   END_RUNG wire#w4
   RUNG wire#w4
      Contact( "Sfty_Commissioning".Udt."200RU01-QQ05_Lock" )
   END_RUNG wire#w5
   RUNG wire#w5
      Contact( "Sfty_Commissioning".Udt."200RU01-BG01_4 _Fence" )
   END_RUNG wire#w6
   RUNG wire#w6
      Contact( "Sfty_Commissioning".Udt.SCH1_SftyLightCurtainDie1 )
   END_RUNG wire#w7
   RUNG wire#w7
      Contact( "Sfty_Commissioning".Udt.SCH1_SftyLightCurtainDie2 )
   END_RUNG wire#w8
   // the same network as SCL:
   #TB1FenceZ200 := ("Sfty_Status"."200RU01-QQ01_Lock".Sig OR "Sfty_Commissioning".Udt."200RU01-QQ01_Lock") AND ("Sfty_Status"."200RU01-QQ02_Lock".Sig OR "Sfty_Commissioning".Udt."200RU01-QQ02_Lock") AND ("Sfty_Status"."200RU01-QQ03_Lock".Sig OR "Sfty_Commissioning".Udt."200RU01-QQ03_Lock") AND ("Sfty_Status"."200RU01-QQ04_Lock".Sig OR "Sfty_Commissioning".Udt."200RU01-QQ04_Lock") AND ("Sfty_Status"."200RU01-QQ05_Lock".Sig OR "Sfty_Commissioning".Udt."200RU01-QQ05_Lock") AND ("Sfty_Status"."200RU01-BG01_4 _Fence".Sig OR "Sfty_Commissioning".Udt."200RU01-BG01_4 _Fence") AND ("Sfty_Comm".SCH1_in.SftyLightCurtainDie1 OR "Sfty_Commissioning".Udt.SCH1_SftyLightCurtainDie1) AND ("Sfty_Comm".SCH1_in.SftyLightCurtainDie2 OR "Sfty_Commissioning".Udt.SCH1_SftyLightCurtainDie2);
END_REGION

REGION Network 13: All doors in zone 300 locked
   RUNG wire#powerrail
      Coil( #TB1FenceZ300 )
   END_RUNG
   // the same network as SCL:
   #TB1FenceZ300 := TRUE;
END_REGION

REGION Network 14: All doors in zone 400 locked
   RUNG wire#powerrail
      Coil( #TB1FenceZ400 )
   END_RUNG
   // the same network as SCL:
   #TB1FenceZ400 := TRUE;
END_REGION

REGION Network 15: *************** Robots section start ***************
END_REGION

REGION Network 16: Safety enable for robots in zone 100
   RUNG wire#powerrail
      Coil( "Sfty_Comm"."1R1+RC01_Out".SftyEn )
   END_RUNG
   RUNG wire#powerrail
      Coil( "Sfty_Comm"."1R2+RC01_Out".SftyEn )
   END_RUNG
   RUNG wire#powerrail
      Coil( "Sfty_Comm"."1R3_4+RC01_Out".SftyEn )
   END_RUNG
   RUNG wire#powerrail
      Coil( "Sfty_Comm"."1R5+RC01_Out".SftyEn )
   END_RUNG
   RUNG wire#powerrail
      Coil( "Sfty_Comm"."1R6+RC01_Out".SftyEn )
   END_RUNG
   // the same network as SCL:
   "Sfty_Comm"."1R1+RC01_Out".SftyEn := TRUE;
   "Sfty_Comm"."1R2+RC01_Out".SftyEn := TRUE;
   "Sfty_Comm"."1R3_4+RC01_Out".SftyEn := TRUE;
   "Sfty_Comm"."1R5+RC01_Out".SftyEn := TRUE;
   "Sfty_Comm"."1R6+RC01_Out".SftyEn := TRUE;
END_REGION

REGION Network 17: Safety enable for robots in zone 200
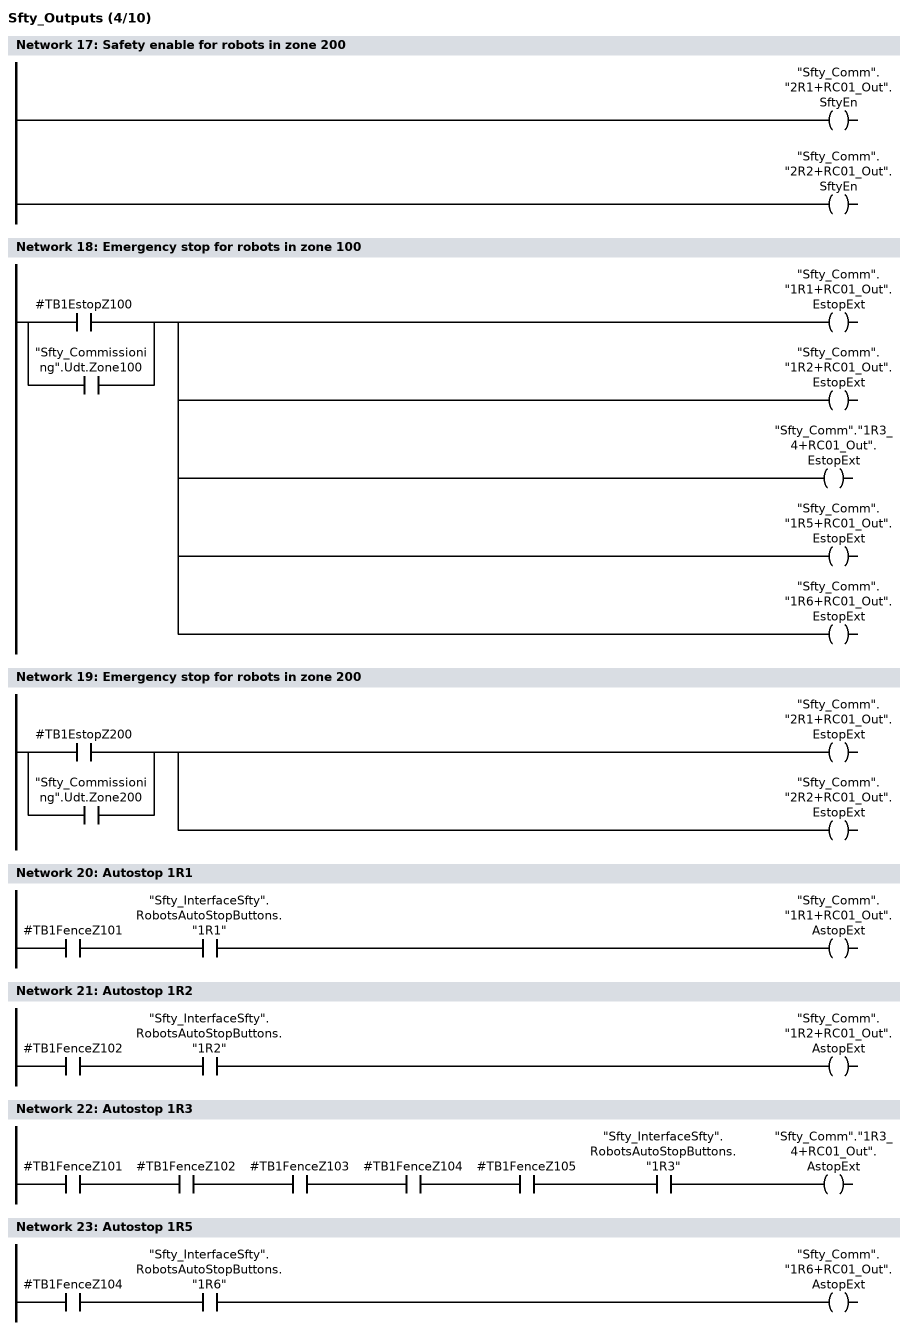
   RUNG wire#powerrail
      Coil( "Sfty_Comm"."2R1+RC01_Out".SftyEn )
   END_RUNG
   RUNG wire#powerrail
      Coil( "Sfty_Comm"."2R2+RC01_Out".SftyEn )
   END_RUNG
   // the same network as SCL:
   "Sfty_Comm"."2R1+RC01_Out".SftyEn := TRUE;
   "Sfty_Comm"."2R2+RC01_Out".SftyEn := TRUE;
END_REGION

REGION Network 18: Emergency stop for robots in zone 100
   RUNG wire#powerrail
      Contact( #TB1EstopZ100 )
      wire#w1
      Coil( "Sfty_Comm"."1R1+RC01_Out".EstopExt )
   END_RUNG
   RUNG wire#powerrail
      Contact( "Sfty_Commissioning".Udt.Zone100 )
   END_RUNG wire#w1
   RUNG wire#w1
      Coil( "Sfty_Comm"."1R2+RC01_Out".EstopExt )
   END_RUNG
   RUNG wire#w1
      Coil( "Sfty_Comm"."1R3_4+RC01_Out".EstopExt )
   END_RUNG
   RUNG wire#w1
      Coil( "Sfty_Comm"."1R5+RC01_Out".EstopExt )
   END_RUNG
   RUNG wire#w1
      Coil( "Sfty_Comm"."1R6+RC01_Out".EstopExt )
   END_RUNG
   // the same network as SCL:
   "Sfty_Comm"."1R1+RC01_Out".EstopExt := #TB1EstopZ100 OR "Sfty_Commissioning".Udt.Zone100;
   "Sfty_Comm"."1R2+RC01_Out".EstopExt := "Sfty_Comm"."1R1+RC01_Out".EstopExt;
   "Sfty_Comm"."1R3_4+RC01_Out".EstopExt := "Sfty_Comm"."1R1+RC01_Out".EstopExt;
   "Sfty_Comm"."1R5+RC01_Out".EstopExt := "Sfty_Comm"."1R1+RC01_Out".EstopExt;
   "Sfty_Comm"."1R6+RC01_Out".EstopExt := "Sfty_Comm"."1R1+RC01_Out".EstopExt;
END_REGION

REGION Network 19: Emergency stop for robots in zone 200
   RUNG wire#powerrail
      Contact( #TB1EstopZ200 )
      wire#w1
      Coil( "Sfty_Comm"."2R1+RC01_Out".EstopExt )
   END_RUNG
   RUNG wire#powerrail
      Contact( "Sfty_Commissioning".Udt.Zone200 )
   END_RUNG wire#w1
   RUNG wire#w1
      Coil( "Sfty_Comm"."2R2+RC01_Out".EstopExt )
   END_RUNG
   // the same network as SCL:
   "Sfty_Comm"."2R1+RC01_Out".EstopExt := #TB1EstopZ200 OR "Sfty_Commissioning".Udt.Zone200;
   "Sfty_Comm"."2R2+RC01_Out".EstopExt := "Sfty_Comm"."2R1+RC01_Out".EstopExt;
END_REGION

REGION Network 20: Autostop 1R1
   RUNG wire#powerrail
      Contact( #TB1FenceZ101 )
      Contact( "Sfty_InterfaceSfty".RobotsAutoStopButtons."1R1" )
      Coil( "Sfty_Comm"."1R1+RC01_Out".AstopExt )
   END_RUNG
   // the same network as SCL:
   "Sfty_Comm"."1R1+RC01_Out".AstopExt := #TB1FenceZ101 AND "Sfty_InterfaceSfty".RobotsAutoStopButtons."1R1";
END_REGION

REGION Network 21: Autostop 1R2
   RUNG wire#powerrail
      Contact( #TB1FenceZ102 )
      Contact( "Sfty_InterfaceSfty".RobotsAutoStopButtons."1R2" )
      Coil( "Sfty_Comm"."1R2+RC01_Out".AstopExt )
   END_RUNG
   // the same network as SCL:
   "Sfty_Comm"."1R2+RC01_Out".AstopExt := #TB1FenceZ102 AND "Sfty_InterfaceSfty".RobotsAutoStopButtons."1R2";
END_REGION

REGION Network 22: Autostop 1R3
   RUNG wire#powerrail
      Contact( #TB1FenceZ101 )
      Contact( #TB1FenceZ102 )
      Contact( #TB1FenceZ103 )
      Contact( #TB1FenceZ104 )
      Contact( #TB1FenceZ105 )
      Contact( "Sfty_InterfaceSfty".RobotsAutoStopButtons."1R3" )
      Coil( "Sfty_Comm"."1R3_4+RC01_Out".AstopExt )
   END_RUNG
   // the same network as SCL:
   "Sfty_Comm"."1R3_4+RC01_Out".AstopExt := #TB1FenceZ101 AND #TB1FenceZ102 AND #TB1FenceZ103 AND #TB1FenceZ104 AND #TB1FenceZ105 AND "Sfty_InterfaceSfty".RobotsAutoStopButtons."1R3";
END_REGION

REGION Network 23: Autostop 1R5
   RUNG wire#powerrail
      Contact( #TB1FenceZ104 )
      Contact( "Sfty_InterfaceSfty".RobotsAutoStopButtons."1R6" )
      Coil( "Sfty_Comm"."1R6+RC01_Out".AstopExt )
   END_RUNG
   // the same network as SCL:
   "Sfty_Comm"."1R6+RC01_Out".AstopExt := #TB1FenceZ104 AND "Sfty_InterfaceSfty".RobotsAutoStopButtons."1R6";
END_REGION

REGION Network 24: Autostop 1R6
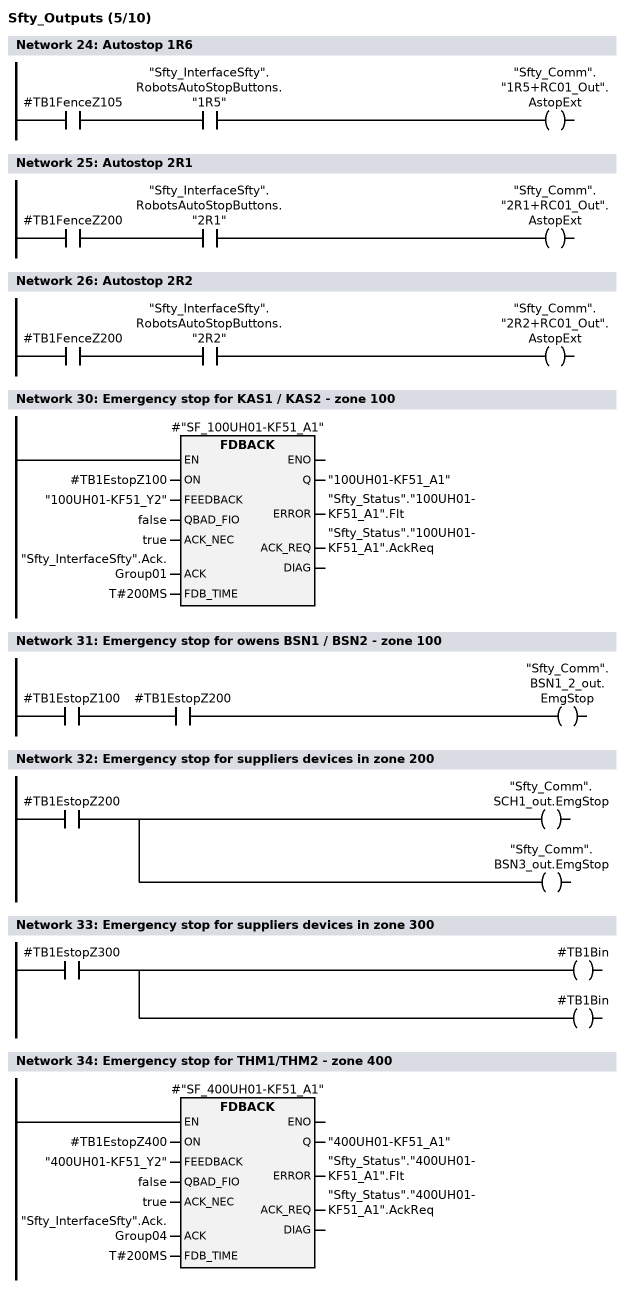
   RUNG wire#powerrail
      Contact( #TB1FenceZ105 )
      Contact( "Sfty_InterfaceSfty".RobotsAutoStopButtons."1R5" )
      Coil( "Sfty_Comm"."1R5+RC01_Out".AstopExt )
   END_RUNG
   // the same network as SCL:
   "Sfty_Comm"."1R5+RC01_Out".AstopExt := #TB1FenceZ105 AND "Sfty_InterfaceSfty".RobotsAutoStopButtons."1R5";
END_REGION

REGION Network 25: Autostop 2R1
   RUNG wire#powerrail
      Contact( #TB1FenceZ200 )
      Contact( "Sfty_InterfaceSfty".RobotsAutoStopButtons."2R1" )
      Coil( "Sfty_Comm"."2R1+RC01_Out".AstopExt )
   END_RUNG
   // the same network as SCL:
   "Sfty_Comm"."2R1+RC01_Out".AstopExt := #TB1FenceZ200 AND "Sfty_InterfaceSfty".RobotsAutoStopButtons."2R1";
END_REGION

REGION Network 26: Autostop 2R2
   RUNG wire#powerrail
      Contact( #TB1FenceZ200 )
      Contact( "Sfty_InterfaceSfty".RobotsAutoStopButtons."2R2" )
      Coil( "Sfty_Comm"."2R2+RC01_Out".AstopExt )
   END_RUNG
   // the same network as SCL:
   "Sfty_Comm"."2R2+RC01_Out".AstopExt := #TB1FenceZ200 AND "Sfty_InterfaceSfty".RobotsAutoStopButtons."2R2";
END_REGION

REGION Network 27: *************** Robots section end ***************
END_REGION

REGION Network 28: *************** Suppliers section start ***************
END_REGION

REGION Network 29: *************** Estop ***************
END_REGION

REGION Network 30: Emergency stop for KAS1 / KAS2 - zone 100
   RUNG wire#powerrail
      #"SF_100UH01-KF51_A1".FDBACK(ON := #TB1EstopZ100, FEEDBACK := "100UH01-KF51_Y2", QBAD_FIO := false, ACK_NEC := true, ACK := "Sfty_InterfaceSfty".Ack.Group01, FDB_TIME := T#200MS, Q => "100UH01-KF51_A1", ERROR => "Sfty_Status"."100UH01-KF51_A1".Flt, ACK_REQ => "Sfty_Status"."100UH01-KF51_A1".AckReq, DIAG =>)
   END_RUNG
   // the same network as SCL:
   #"SF_100UH01-KF51_A1"(ON := #TB1EstopZ100,   // FDBACK
                         FEEDBACK := "100UH01-KF51_Y2",
                         QBAD_FIO := false,
                         ACK_NEC := true,
                         ACK := "Sfty_InterfaceSfty".Ack.Group01,
                         FDB_TIME := T#200MS,
                         Q => "100UH01-KF51_A1",
                         ERROR => "Sfty_Status"."100UH01-KF51_A1".Flt,
                         ACK_REQ => "Sfty_Status"."100UH01-KF51_A1".AckReq);
END_REGION

REGION Network 31: Emergency stop for owens BSN1 / BSN2 - zone 100
   RUNG wire#powerrail
      Contact( #TB1EstopZ100 )
      Contact( #TB1EstopZ200 )
      Coil( "Sfty_Comm".BSN1_2_out.EmgStop )
   END_RUNG
   // the same network as SCL:
   "Sfty_Comm".BSN1_2_out.EmgStop := #TB1EstopZ100 AND #TB1EstopZ200;
END_REGION

REGION Network 32: Emergency stop for suppliers devices in zone 200
   RUNG wire#powerrail
      Contact( #TB1EstopZ200 )
      wire#w1
      Coil( "Sfty_Comm".SCH1_out.EmgStop )
   END_RUNG
   RUNG wire#w1
      Coil( "Sfty_Comm".BSN3_out.EmgStop )
   END_RUNG
   // the same network as SCL:
   "Sfty_Comm".SCH1_out.EmgStop := #TB1EstopZ200;
   "Sfty_Comm".BSN3_out.EmgStop := #TB1EstopZ200;
END_REGION

REGION Network 33: Emergency stop for suppliers devices in zone 300
   RUNG wire#powerrail
      Contact( #TB1EstopZ300 )
      wire#w1
      Coil( #TB1Bin )
   END_RUNG
   RUNG wire#w1
      Coil( #TB1Bin )
   END_RUNG
   // the same network as SCL:
   #TB1Bin := #TB1EstopZ300;
   #TB1Bin := #TB1EstopZ300;
END_REGION

REGION Network 34: Emergency stop for THM1/THM2 - zone 400
   RUNG wire#powerrail
      #"SF_400UH01-KF51_A1".FDBACK(ON := #TB1EstopZ400, FEEDBACK := "400UH01-KF51_Y2", QBAD_FIO := false, ACK_NEC := true, ACK := "Sfty_InterfaceSfty".Ack.Group04, FDB_TIME := T#200MS, Q => "400UH01-KF51_A1", ERROR => "Sfty_Status"."400UH01-KF51_A1".Flt, ACK_REQ => "Sfty_Status"."400UH01-KF51_A1".AckReq, DIAG =>)
   END_RUNG
   // the same network as SCL:
   #"SF_400UH01-KF51_A1"(ON := #TB1EstopZ400,   // FDBACK
                         FEEDBACK := "400UH01-KF51_Y2",
                         QBAD_FIO := false,
                         ACK_NEC := true,
                         ACK := "Sfty_InterfaceSfty".Ack.Group04,
                         FDB_TIME := T#200MS,
                         Q => "400UH01-KF51_A1",
                         ERROR => "Sfty_Status"."400UH01-KF51_A1".Flt,
                         ACK_REQ => "Sfty_Status"."400UH01-KF51_A1".AckReq);
END_REGION

REGION Network 35: Emergency stop for suppliers devices in zone 400
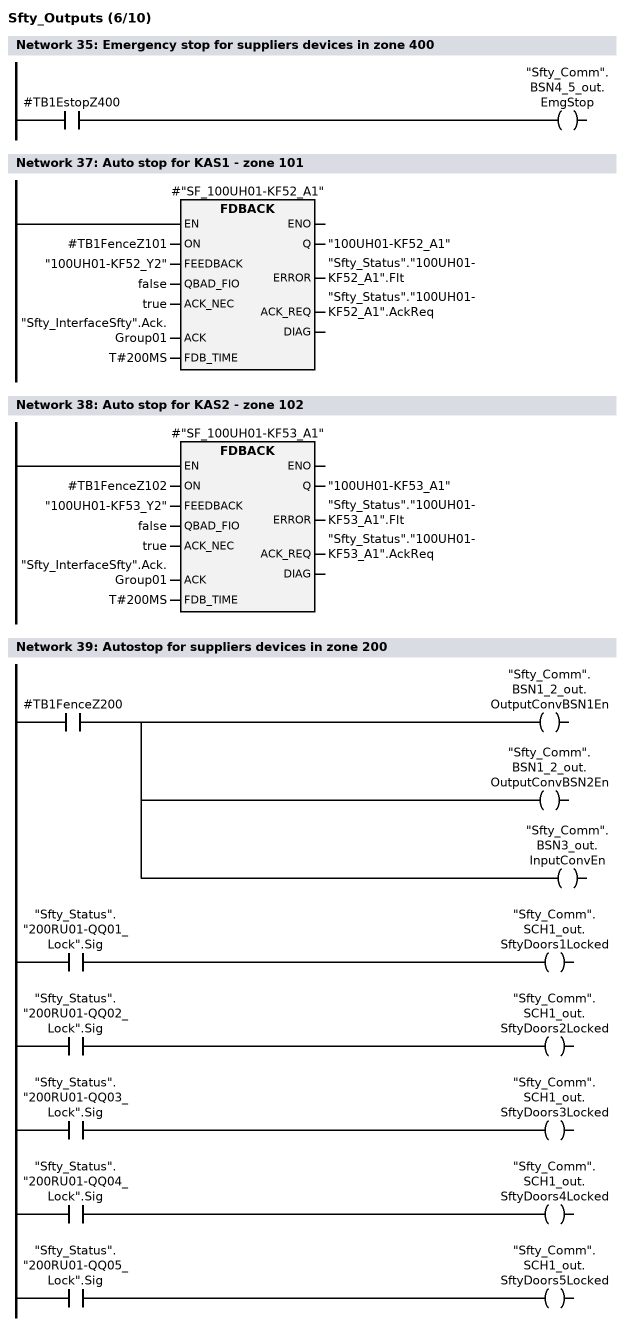
   RUNG wire#powerrail
      Contact( #TB1EstopZ400 )
      Coil( "Sfty_Comm".BSN4_5_out.EmgStop )
   END_RUNG
   // the same network as SCL:
   "Sfty_Comm".BSN4_5_out.EmgStop := #TB1EstopZ400;
END_REGION

REGION Network 36: *************** Auto stop ***************
END_REGION

REGION Network 37: Auto stop for KAS1 - zone 101
   RUNG wire#powerrail
      #"SF_100UH01-KF52_A1".FDBACK(ON := #TB1FenceZ101, FEEDBACK := "100UH01-KF52_Y2", QBAD_FIO := false, ACK_NEC := true, ACK := "Sfty_InterfaceSfty".Ack.Group01, FDB_TIME := T#200MS, Q => "100UH01-KF52_A1", ERROR => "Sfty_Status"."100UH01-KF52_A1".Flt, ACK_REQ => "Sfty_Status"."100UH01-KF52_A1".AckReq, DIAG =>)
   END_RUNG
   // the same network as SCL:
   #"SF_100UH01-KF52_A1"(ON := #TB1FenceZ101,   // FDBACK
                         FEEDBACK := "100UH01-KF52_Y2",
                         QBAD_FIO := false,
                         ACK_NEC := true,
                         ACK := "Sfty_InterfaceSfty".Ack.Group01,
                         FDB_TIME := T#200MS,
                         Q => "100UH01-KF52_A1",
                         ERROR => "Sfty_Status"."100UH01-KF52_A1".Flt,
                         ACK_REQ => "Sfty_Status"."100UH01-KF52_A1".AckReq);
END_REGION

REGION Network 38: Auto stop for KAS2 - zone 102
   RUNG wire#powerrail
      #"SF_100UH01-KF53_A1".FDBACK(ON := #TB1FenceZ102, FEEDBACK := "100UH01-KF53_Y2", QBAD_FIO := false, ACK_NEC := true, ACK := "Sfty_InterfaceSfty".Ack.Group01, FDB_TIME := T#200MS, Q => "100UH01-KF53_A1", ERROR => "Sfty_Status"."100UH01-KF53_A1".Flt, ACK_REQ => "Sfty_Status"."100UH01-KF53_A1".AckReq, DIAG =>)
   END_RUNG
   // the same network as SCL:
   #"SF_100UH01-KF53_A1"(ON := #TB1FenceZ102,   // FDBACK
                         FEEDBACK := "100UH01-KF53_Y2",
                         QBAD_FIO := false,
                         ACK_NEC := true,
                         ACK := "Sfty_InterfaceSfty".Ack.Group01,
                         FDB_TIME := T#200MS,
                         Q => "100UH01-KF53_A1",
                         ERROR => "Sfty_Status"."100UH01-KF53_A1".Flt,
                         ACK_REQ => "Sfty_Status"."100UH01-KF53_A1".AckReq);
END_REGION

REGION Network 39: Autostop for suppliers devices in zone 200
   RUNG wire#powerrail
      Contact( #TB1FenceZ200 )
      wire#w1
      Coil( "Sfty_Comm".BSN1_2_out.OutputConvBSN1En )
   END_RUNG
   RUNG wire#w1
      Coil( "Sfty_Comm".BSN1_2_out.OutputConvBSN2En )
   END_RUNG
   RUNG wire#w1
      Coil( "Sfty_Comm".BSN3_out.InputConvEn )
   END_RUNG
   RUNG wire#powerrail
      Contact( "Sfty_Status"."200RU01-QQ01_Lock".Sig )
      Coil( "Sfty_Comm".SCH1_out.SftyDoors1Locked )
   END_RUNG
   RUNG wire#powerrail
      Contact( "Sfty_Status"."200RU01-QQ02_Lock".Sig )
      Coil( "Sfty_Comm".SCH1_out.SftyDoors2Locked )
   END_RUNG
   RUNG wire#powerrail
      Contact( "Sfty_Status"."200RU01-QQ03_Lock".Sig )
      Coil( "Sfty_Comm".SCH1_out.SftyDoors3Locked )
   END_RUNG
   RUNG wire#powerrail
      Contact( "Sfty_Status"."200RU01-QQ04_Lock".Sig )
      Coil( "Sfty_Comm".SCH1_out.SftyDoors4Locked )
   END_RUNG
   RUNG wire#powerrail
      Contact( "Sfty_Status"."200RU01-QQ05_Lock".Sig )
      Coil( "Sfty_Comm".SCH1_out.SftyDoors5Locked )
   END_RUNG
   // the same network as SCL:
   "Sfty_Comm".BSN1_2_out.OutputConvBSN1En := #TB1FenceZ200;
   "Sfty_Comm".BSN1_2_out.OutputConvBSN2En := #TB1FenceZ200;
   "Sfty_Comm".BSN3_out.InputConvEn := #TB1FenceZ200;
   "Sfty_Comm".SCH1_out.SftyDoors1Locked := "Sfty_Status"."200RU01-QQ01_Lock".Sig;
   "Sfty_Comm".SCH1_out.SftyDoors2Locked := "Sfty_Status"."200RU01-QQ02_Lock".Sig;
   "Sfty_Comm".SCH1_out.SftyDoors3Locked := "Sfty_Status"."200RU01-QQ03_Lock".Sig;
   "Sfty_Comm".SCH1_out.SftyDoors4Locked := "Sfty_Status"."200RU01-QQ04_Lock".Sig;
   "Sfty_Comm".SCH1_out.SftyDoors5Locked := "Sfty_Status"."200RU01-QQ05_Lock".Sig;
END_REGION

REGION Network 40: Autostop for suppliers devices in zone 300
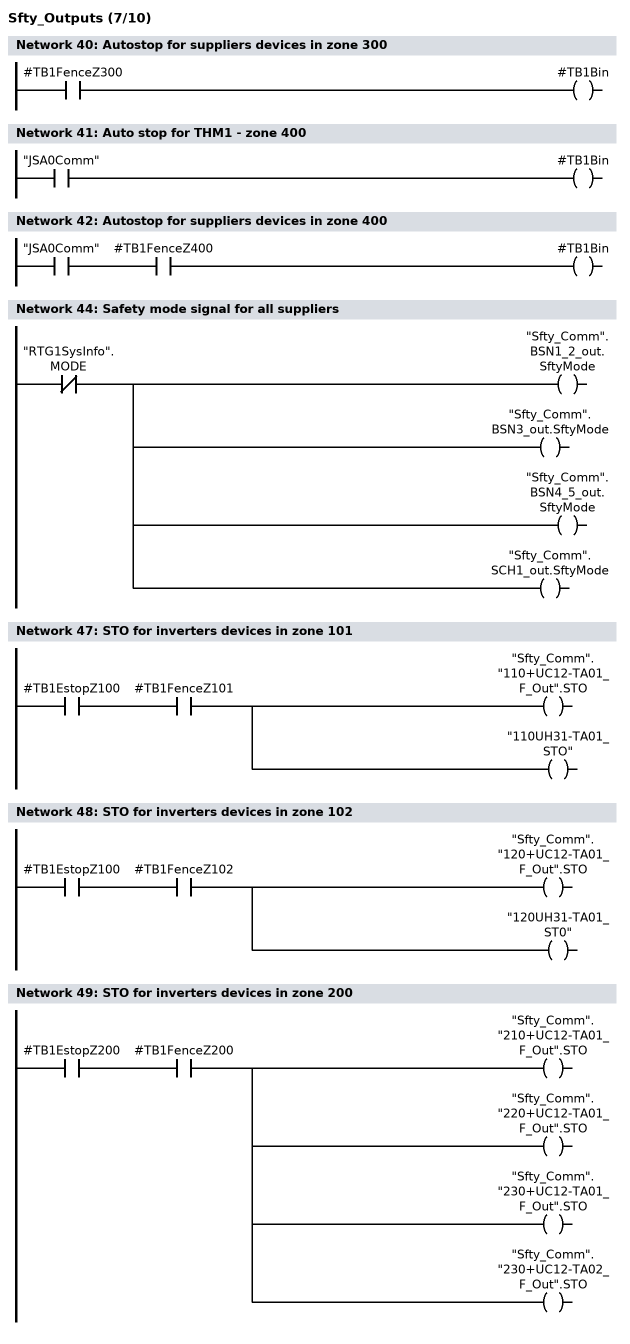
   RUNG wire#powerrail
      Contact( #TB1FenceZ300 )
      Coil( #TB1Bin )
   END_RUNG
   // the same network as SCL:
   #TB1Bin := #TB1FenceZ300;
END_REGION

REGION Network 41: Auto stop for THM1 - zone 400
   RUNG wire#powerrail
      Contact( "JSA0Comm" )
      Coil( #TB1Bin )
   END_RUNG
   // the same network as SCL:
   #TB1Bin := "JSA0Comm";
END_REGION

REGION Network 42: Autostop for suppliers devices in zone 400
   RUNG wire#powerrail
      Contact( "JSA0Comm" )
      Contact( #TB1FenceZ400 )
      Coil( #TB1Bin )
   END_RUNG
   // the same network as SCL:
   #TB1Bin := "JSA0Comm" AND #TB1FenceZ400;
END_REGION

REGION Network 43: *************** Safety mode ***************
END_REGION

REGION Network 44: Safety mode signal for all suppliers
   RUNG wire#powerrail
      I_Contact( "RTG1SysInfo".MODE )
      wire#w1
      Coil( "Sfty_Comm".BSN1_2_out.SftyMode )
   END_RUNG
   RUNG wire#w1
      Coil( "Sfty_Comm".BSN3_out.SftyMode )
   END_RUNG
   RUNG wire#w1
      Coil( "Sfty_Comm".BSN4_5_out.SftyMode )
   END_RUNG
   RUNG wire#w1
      Coil( "Sfty_Comm".SCH1_out.SftyMode )
   END_RUNG
   // the same network as SCL:
   "Sfty_Comm".BSN1_2_out.SftyMode := NOT "RTG1SysInfo".MODE;
   "Sfty_Comm".BSN3_out.SftyMode := NOT "RTG1SysInfo".MODE;
   "Sfty_Comm".BSN4_5_out.SftyMode := NOT "RTG1SysInfo".MODE;
   "Sfty_Comm".SCH1_out.SftyMode := NOT "RTG1SysInfo".MODE;
END_REGION

REGION Network 45: *************** Suppliers section end ***************
END_REGION

REGION Network 46: *************** Inverters section start ***************
END_REGION

REGION Network 47: STO for inverters devices in zone 101
   RUNG wire#powerrail
      Contact( #TB1EstopZ100 )
      Contact( #TB1FenceZ101 )
      wire#w1
      Coil( "Sfty_Comm"."110+UC12-TA01_F_Out".STO )
   END_RUNG
   RUNG wire#w1
      Coil( "110UH31-TA01_STO" )
   END_RUNG
   // the same network as SCL:
   "Sfty_Comm"."110+UC12-TA01_F_Out".STO := #TB1EstopZ100 AND #TB1FenceZ101;
   "110UH31-TA01_STO" := "Sfty_Comm"."110+UC12-TA01_F_Out".STO;
END_REGION

REGION Network 48: STO for inverters devices in zone 102
   RUNG wire#powerrail
      Contact( #TB1EstopZ100 )
      Contact( #TB1FenceZ102 )
      wire#w1
      Coil( "Sfty_Comm"."120+UC12-TA01_F_Out".STO )
   END_RUNG
   RUNG wire#w1
      Coil( "120UH31-TA01_ST0" )
   END_RUNG
   // the same network as SCL:
   "Sfty_Comm"."120+UC12-TA01_F_Out".STO := #TB1EstopZ100 AND #TB1FenceZ102;
   "120UH31-TA01_ST0" := "Sfty_Comm"."120+UC12-TA01_F_Out".STO;
END_REGION

REGION Network 49: STO for inverters devices in zone 200
   RUNG wire#powerrail
      Contact( #TB1EstopZ200 )
      Contact( #TB1FenceZ200 )
      wire#w1
      Coil( "Sfty_Comm"."210+UC12-TA01_F_Out".STO )
   END_RUNG
   RUNG wire#w1
      Coil( "Sfty_Comm"."220+UC12-TA01_F_Out".STO )
   END_RUNG
   RUNG wire#w1
      Coil( "Sfty_Comm"."230+UC12-TA01_F_Out".STO )
   END_RUNG
   RUNG wire#w1
      Coil( "Sfty_Comm"."230+UC12-TA02_F_Out".STO )
   END_RUNG
   // the same network as SCL:
   "Sfty_Comm"."210+UC12-TA01_F_Out".STO := #TB1EstopZ200 AND #TB1FenceZ200;
   "Sfty_Comm"."220+UC12-TA01_F_Out".STO := "Sfty_Comm"."210+UC12-TA01_F_Out".STO;
   "Sfty_Comm"."230+UC12-TA01_F_Out".STO := "Sfty_Comm"."210+UC12-TA01_F_Out".STO;
   "Sfty_Comm"."230+UC12-TA02_F_Out".STO := "Sfty_Comm"."210+UC12-TA01_F_Out".STO;
END_REGION

REGION Network 50: STO for inverters devices in zone 300
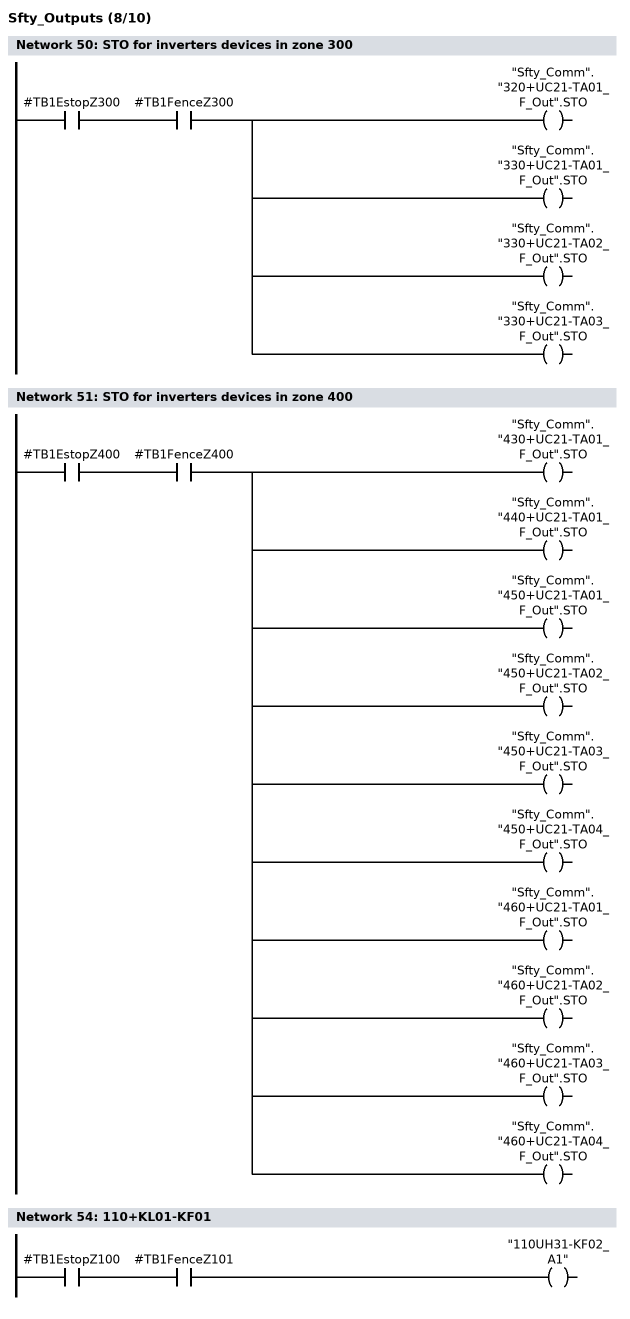
   RUNG wire#powerrail
      Contact( #TB1EstopZ300 )
      Contact( #TB1FenceZ300 )
      wire#w1
      Coil( "Sfty_Comm"."320+UC21-TA01_F_Out".STO )
   END_RUNG
   RUNG wire#w1
      Coil( "Sfty_Comm"."330+UC21-TA01_F_Out".STO )
   END_RUNG
   RUNG wire#w1
      Coil( "Sfty_Comm"."330+UC21-TA02_F_Out".STO )
   END_RUNG
   RUNG wire#w1
      Coil( "Sfty_Comm"."330+UC21-TA03_F_Out".STO )
   END_RUNG
   // the same network as SCL:
   "Sfty_Comm"."320+UC21-TA01_F_Out".STO := #TB1EstopZ300 AND #TB1FenceZ300;
   "Sfty_Comm"."330+UC21-TA01_F_Out".STO := "Sfty_Comm"."320+UC21-TA01_F_Out".STO;
   "Sfty_Comm"."330+UC21-TA02_F_Out".STO := "Sfty_Comm"."320+UC21-TA01_F_Out".STO;
   "Sfty_Comm"."330+UC21-TA03_F_Out".STO := "Sfty_Comm"."320+UC21-TA01_F_Out".STO;
END_REGION

REGION Network 51: STO for inverters devices in zone 400
   RUNG wire#powerrail
      Contact( #TB1EstopZ400 )
      Contact( #TB1FenceZ400 )
      wire#w1
      Coil( "Sfty_Comm"."430+UC21-TA01_F_Out".STO )
   END_RUNG
   RUNG wire#w1
      Coil( "Sfty_Comm"."440+UC21-TA01_F_Out".STO )
   END_RUNG
   RUNG wire#w1
      Coil( "Sfty_Comm"."450+UC21-TA01_F_Out".STO )
   END_RUNG
   RUNG wire#w1
      Coil( "Sfty_Comm"."450+UC21-TA02_F_Out".STO )
   END_RUNG
   RUNG wire#w1
      Coil( "Sfty_Comm"."450+UC21-TA03_F_Out".STO )
   END_RUNG
   RUNG wire#w1
      Coil( "Sfty_Comm"."450+UC21-TA04_F_Out".STO )
   END_RUNG
   RUNG wire#w1
      Coil( "Sfty_Comm"."460+UC21-TA01_F_Out".STO )
   END_RUNG
   RUNG wire#w1
      Coil( "Sfty_Comm"."460+UC21-TA02_F_Out".STO )
   END_RUNG
   RUNG wire#w1
      Coil( "Sfty_Comm"."460+UC21-TA03_F_Out".STO )
   END_RUNG
   RUNG wire#w1
      Coil( "Sfty_Comm"."460+UC21-TA04_F_Out".STO )
   END_RUNG
   // the same network as SCL:
   "Sfty_Comm"."430+UC21-TA01_F_Out".STO := #TB1EstopZ400 AND #TB1FenceZ400;
   "Sfty_Comm"."440+UC21-TA01_F_Out".STO := "Sfty_Comm"."430+UC21-TA01_F_Out".STO;
   "Sfty_Comm"."450+UC21-TA01_F_Out".STO := "Sfty_Comm"."430+UC21-TA01_F_Out".STO;
   "Sfty_Comm"."450+UC21-TA02_F_Out".STO := "Sfty_Comm"."430+UC21-TA01_F_Out".STO;
   "Sfty_Comm"."450+UC21-TA03_F_Out".STO := "Sfty_Comm"."430+UC21-TA01_F_Out".STO;
   "Sfty_Comm"."450+UC21-TA04_F_Out".STO := "Sfty_Comm"."430+UC21-TA01_F_Out".STO;
   "Sfty_Comm"."460+UC21-TA01_F_Out".STO := "Sfty_Comm"."430+UC21-TA01_F_Out".STO;
   "Sfty_Comm"."460+UC21-TA02_F_Out".STO := "Sfty_Comm"."430+UC21-TA01_F_Out".STO;
   "Sfty_Comm"."460+UC21-TA03_F_Out".STO := "Sfty_Comm"."430+UC21-TA01_F_Out".STO;
   "Sfty_Comm"."460+UC21-TA04_F_Out".STO := "Sfty_Comm"."430+UC21-TA01_F_Out".STO;
END_REGION

REGION Network 52: *************** Inverters section end ***************
END_REGION

REGION Network 53: *************** Valve terminals section start ***************
END_REGION

REGION Network 54: 110+KL01-KF01
   RUNG wire#powerrail
      Contact( #TB1EstopZ100 )
      Contact( #TB1FenceZ101 )
      Coil( "110UH31-KF02_A1" )
   END_RUNG
   // the same network as SCL:
   "110UH31-KF02_A1" := #TB1EstopZ100 AND #TB1FenceZ101;
END_REGION

REGION Network 55: 120+KL01-KF01
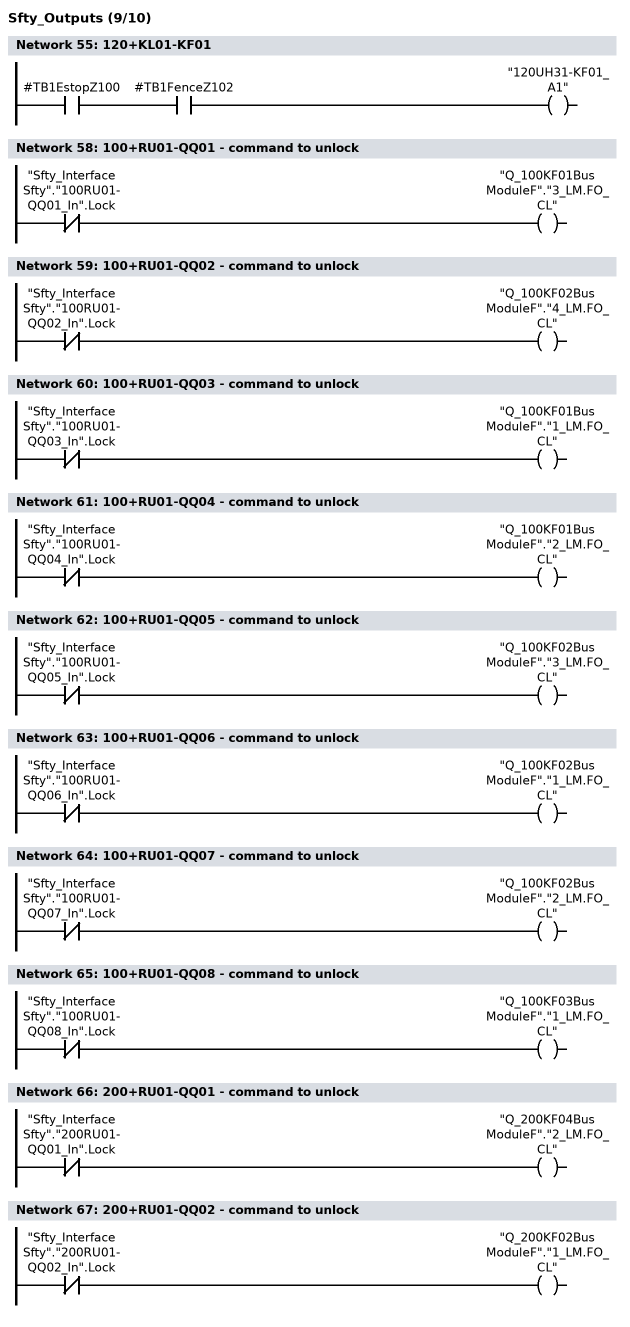
   RUNG wire#powerrail
      Contact( #TB1EstopZ100 )
      Contact( #TB1FenceZ102 )
      Coil( "120UH31-KF01_A1" )
   END_RUNG
   // the same network as SCL:
   "120UH31-KF01_A1" := #TB1EstopZ100 AND #TB1FenceZ102;
END_REGION

REGION Network 56: *************** Valve terminals section end ***************
END_REGION

REGION Network 57: *************** Unlock gates commands section start ***************
END_REGION

REGION Network 58: 100+RU01-QQ01 - command to unlock
   RUNG wire#powerrail
      I_Contact( "Sfty_InterfaceSfty"."100RU01-QQ01_In".Lock )
      Coil( "Q_100KF01BusModuleF"."3_LM.FO_CL" )
   END_RUNG
   // the same network as SCL:
   "Q_100KF01BusModuleF"."3_LM.FO_CL" := NOT "Sfty_InterfaceSfty"."100RU01-QQ01_In".Lock;
END_REGION

REGION Network 59: 100+RU01-QQ02 - command to unlock
   RUNG wire#powerrail
      I_Contact( "Sfty_InterfaceSfty"."100RU01-QQ02_In".Lock )
      Coil( "Q_100KF02BusModuleF"."4_LM.FO_CL" )
   END_RUNG
   // the same network as SCL:
   "Q_100KF02BusModuleF"."4_LM.FO_CL" := NOT "Sfty_InterfaceSfty"."100RU01-QQ02_In".Lock;
END_REGION

REGION Network 60: 100+RU01-QQ03 - command to unlock
   RUNG wire#powerrail
      I_Contact( "Sfty_InterfaceSfty"."100RU01-QQ03_In".Lock )
      Coil( "Q_100KF01BusModuleF"."1_LM.FO_CL" )
   END_RUNG
   // the same network as SCL:
   "Q_100KF01BusModuleF"."1_LM.FO_CL" := NOT "Sfty_InterfaceSfty"."100RU01-QQ03_In".Lock;
END_REGION

REGION Network 61: 100+RU01-QQ04 - command to unlock
   RUNG wire#powerrail
      I_Contact( "Sfty_InterfaceSfty"."100RU01-QQ04_In".Lock )
      Coil( "Q_100KF01BusModuleF"."2_LM.FO_CL" )
   END_RUNG
   // the same network as SCL:
   "Q_100KF01BusModuleF"."2_LM.FO_CL" := NOT "Sfty_InterfaceSfty"."100RU01-QQ04_In".Lock;
END_REGION

REGION Network 62: 100+RU01-QQ05 - command to unlock
   RUNG wire#powerrail
      I_Contact( "Sfty_InterfaceSfty"."100RU01-QQ05_In".Lock )
      Coil( "Q_100KF02BusModuleF"."3_LM.FO_CL" )
   END_RUNG
   // the same network as SCL:
   "Q_100KF02BusModuleF"."3_LM.FO_CL" := NOT "Sfty_InterfaceSfty"."100RU01-QQ05_In".Lock;
END_REGION

REGION Network 63: 100+RU01-QQ06 - command to unlock
   RUNG wire#powerrail
      I_Contact( "Sfty_InterfaceSfty"."100RU01-QQ06_In".Lock )
      Coil( "Q_100KF02BusModuleF"."1_LM.FO_CL" )
   END_RUNG
   // the same network as SCL:
   "Q_100KF02BusModuleF"."1_LM.FO_CL" := NOT "Sfty_InterfaceSfty"."100RU01-QQ06_In".Lock;
END_REGION

REGION Network 64: 100+RU01-QQ07 - command to unlock
   RUNG wire#powerrail
      I_Contact( "Sfty_InterfaceSfty"."100RU01-QQ07_In".Lock )
      Coil( "Q_100KF02BusModuleF"."2_LM.FO_CL" )
   END_RUNG
   // the same network as SCL:
   "Q_100KF02BusModuleF"."2_LM.FO_CL" := NOT "Sfty_InterfaceSfty"."100RU01-QQ07_In".Lock;
END_REGION

REGION Network 65: 100+RU01-QQ08 - command to unlock
   RUNG wire#powerrail
      I_Contact( "Sfty_InterfaceSfty"."100RU01-QQ08_In".Lock )
      Coil( "Q_100KF03BusModuleF"."1_LM.FO_CL" )
   END_RUNG
   // the same network as SCL:
   "Q_100KF03BusModuleF"."1_LM.FO_CL" := NOT "Sfty_InterfaceSfty"."100RU01-QQ08_In".Lock;
END_REGION

REGION Network 66: 200+RU01-QQ01 - command to unlock
   RUNG wire#powerrail
      I_Contact( "Sfty_InterfaceSfty"."200RU01-QQ01_In".Lock )
      Coil( "Q_200KF04BusModuleF"."2_LM.FO_CL" )
   END_RUNG
   // the same network as SCL:
   "Q_200KF04BusModuleF"."2_LM.FO_CL" := NOT "Sfty_InterfaceSfty"."200RU01-QQ01_In".Lock;
END_REGION

REGION Network 67: 200+RU01-QQ02 - command to unlock
   RUNG wire#powerrail
      I_Contact( "Sfty_InterfaceSfty"."200RU01-QQ02_In".Lock )
      Coil( "Q_200KF02BusModuleF"."1_LM.FO_CL" )
   END_RUNG
   // the same network as SCL:
   "Q_200KF02BusModuleF"."1_LM.FO_CL" := NOT "Sfty_InterfaceSfty"."200RU01-QQ02_In".Lock;
END_REGION

REGION Network 68: 200+RU01-QQ03 - command to unlock
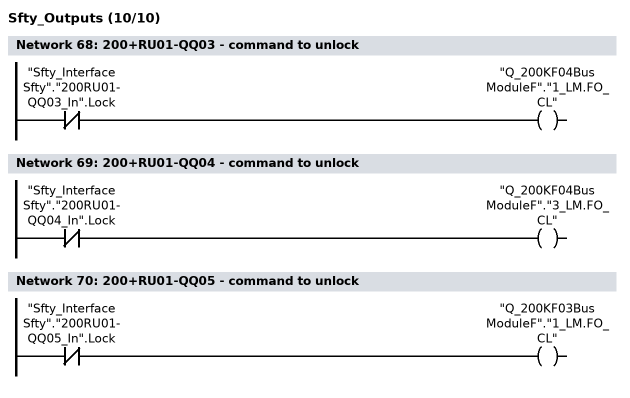
   RUNG wire#powerrail
      I_Contact( "Sfty_InterfaceSfty"."200RU01-QQ03_In".Lock )
      Coil( "Q_200KF04BusModuleF"."1_LM.FO_CL" )
   END_RUNG
   // the same network as SCL:
   "Q_200KF04BusModuleF"."1_LM.FO_CL" := NOT "Sfty_InterfaceSfty"."200RU01-QQ03_In".Lock;
END_REGION

REGION Network 69: 200+RU01-QQ04 - command to unlock
   RUNG wire#powerrail
      I_Contact( "Sfty_InterfaceSfty"."200RU01-QQ04_In".Lock )
      Coil( "Q_200KF04BusModuleF"."3_LM.FO_CL" )
   END_RUNG
   // the same network as SCL:
   "Q_200KF04BusModuleF"."3_LM.FO_CL" := NOT "Sfty_InterfaceSfty"."200RU01-QQ04_In".Lock;
END_REGION

REGION Network 70: 200+RU01-QQ05 - command to unlock
   RUNG wire#powerrail
      I_Contact( "Sfty_InterfaceSfty"."200RU01-QQ05_In".Lock )
      Coil( "Q_200KF03BusModuleF"."1_LM.FO_CL" )
   END_RUNG
   // the same network as SCL:
   "Q_200KF03BusModuleF"."1_LM.FO_CL" := NOT "Sfty_InterfaceSfty"."200RU01-QQ05_In".Lock;
END_REGION

REGION Network 71: *************** Unlock gates commands section end ***************
END_REGION
END_FUNCTION_BLOCK
